    !************************************************
    ! Function    :     Initialize Variables
    ! Programmer  :     Philippe Fleischmann
    ! Date        :     2019.02.22
    !***************** ETH Zurich *******************
    !
    PROC r_RRC_InitVar()
        !
        ! Set Task on
        b_RRC_TaskReceiverOn:=TRUE;
        !
        ! Reset buffer full bits controller
        b_RRC_BufFullMa{n_RRC_R1_ChaNr}:=FALSE;
        b_RRC_BufFullMa{n_RRC_R2_ChaNr}:=FALSE;
        b_RRC_BufFullMa{n_RRC_R3_ChaNr}:=FALSE;
        b_RRC_BufFullMa{n_RRC_R4_ChaNr}:=FALSE;
        !
        ! Reset buffer full bits robot
        b_RRC_BufFullRob{n_RRC_R1_ChaNr}:=FALSE;
        b_RRC_BufFullRob{n_RRC_R2_ChaNr}:=FALSE;
        b_RRC_BufFullRob{n_RRC_R3_ChaNr}:=FALSE;
        b_RRC_BufFullRob{n_RRC_R4_ChaNr}:=FALSE;
        !
        ! Set first cycle bools
        b_RRC_FirstProtocolAfterPPMain:=TRUE;
        !
        ! Temp to measure cycle time
        b_RRC_FeedbackOut:=FALSE;
        !
        ! Reset counters controller
        n_RRC_WritePtrBufCtrl{n_RRC_R1_ChaNr}:=0;
        n_RRC_WritePtrBufCtrl{n_RRC_R2_ChaNr}:=0;
        n_RRC_WritePtrBufCtrl{n_RRC_R3_ChaNr}:=0;
        n_RRC_WritePtrBufCtrl{n_RRC_R4_ChaNr}:=0;
        !
        ! Reset counters robot
        n_RRC_WritePtrBufRob{n_RRC_R1_ChaNr}:=0;
        n_RRC_WritePtrBufRob{n_RRC_R2_ChaNr}:=0;
        n_RRC_WritePtrBufRob{n_RRC_R3_ChaNr}:=0;
        n_RRC_WritePtrBufRob{n_RRC_R4_ChaNr}:=0;
        !
        ! Clear buffer controller
        FOR i FROM 1 TO DIM(bm_RRC_RecBufferCtrl,2) DO
            !
            ! Overwrite with an empty message
            bm_RRC_RecBufferCtrl{n_RRC_R1_ChaNr,i}:=bmEmpty;
            bm_RRC_RecBufferCtrl{n_RRC_R2_ChaNr,i}:=bmEmpty;
            bm_RRC_RecBufferCtrl{n_RRC_R3_ChaNr,i}:=bmEmpty;
            bm_RRC_RecBufferCtrl{n_RRC_R4_ChaNr,i}:=bmEmpty;
            !
        ENDFOR
        !
        ! Clear buffer robots
        FOR i FROM 1 TO DIM(bm_RRC_RecBufferRob,2) DO
            !
            ! Overwrite with an empty message
            bm_RRC_RecBufferRob{n_RRC_R1_ChaNr,i}:=bmEmpty;
            bm_RRC_RecBufferRob{n_RRC_R2_ChaNr,i}:=bmEmpty;
            bm_RRC_RecBufferRob{n_RRC_R3_ChaNr,i}:=bmEmpty;
            bm_RRC_RecBufferRob{n_RRC_R4_ChaNr,i}:=bmEmpty;
            !
        ENDFOR
        !
        ! Reset expected Sequince ID
        n_RRC_SIDExpected{n_RRC_R1_ChaNr}:=0;
        n_RRC_SIDExpected{n_RRC_R2_ChaNr}:=0;
        n_RRC_SIDExpected{n_RRC_R3_ChaNr}:=0;
        n_RRC_SIDExpected{n_RRC_R4_ChaNr}:=0;
        RETURN ;
    ERROR
        ! Placeholder for Error Code...
    ENDPROC

    !************************************************
    ! Function    :     ProgError
    ! Programmer  :     Philippe Fleischmann
    ! Date        :     2019.02.22
    !***************** ETH Zurich *******************
    !
    PROC r_RRC_ProgError()
        !
        ! User Info
        TPWrite "Program Error";
        !
        ! Stop Program
        Stop;
        RETURN ;
    ERROR
        ! Placeholder for Error Code...
    ENDPROC

ENDMODULE

--- Controller Data/v2600-510970_CAADRIA/RAPID/TASK3/SYSMOD/RRC_DataTask_Rx.sys ---
MODULE RRC_DataTask_Rx(SYSMODULE)
    !***********************************************************************************
    !
    ! ETH Zurich / Robotic Fabrication Lab
    ! HIB C 13 / Stefano-Franscini-Platz 1
    ! CH-8093 Zurich
    !
    !***********************************************************************************
    !
    ! PROJECT     :  RRC - Rapid Robot Communication
    !
    ! FUNCTION    :  Includ all Task specific Data's
    !
    ! AUTHOR      :  Philippe Fleischmann
    !
    ! EMAIL       :  rrc@arch.ethz.ch
    !
    ! HISTORY     :  2019.02.22
    !
    ! Copyright   :  ETH Zurich (CH) 2019
    !                - Philippe Fleischmann
    !                - Michael Lyrenmann
    !                - Gonzalo Casas
    !
    ! License     :  This code base is governed by an EULA (End-User License Agreement)
    !                which you have received together with the software.
    !                You are not allowed to use the software on a real robots
    !                without a signed EULA.
    !
    !                A copy of the EULA content is in the controller task (T_CTRL).
    !
    !***********************************************************************************

    !************************************************
    ! Declaration :     bool
    !************************************************
    !
    CONST bool b_RRC_Run:=TRUE;
    !
    TASK PERS bool b_RRC_SocketActiv:=TRUE;
    TASK PERS bool b_RRC_PrintPrio1:=FALSE;
    TASK PERS bool b_RRC_PrintPrio2:=FALSE;
    !
    TASK PERS bool b_RRC_BufFullMa{n_RRC_NumOfCha}:=[FALSE,FALSE,FALSE,FALSE];
    TASK PERS bool b_RRC_BufFullRob{n_RRC_NumOfCha}:=[FALSE,FALSE,FALSE,FALSE];
    TASK PERS bool b_RRC_LogHelper{n_RRC_NumOfCha}:=[FALSE,FALSE,FALSE,FALSE];
    !
    TASK PERS bool b_RRC_FirstProtocolAfterPPMain:=FALSE;

    !************************************************
    ! Declaration :     num
    !************************************************
    !
    CONST num n_RRC_NumOfCha:=4;
    CONST num n_RRC_RecMinData:=49;
    CONST num n_RRC_NoOfByMsgLen:=4;
    CONST num n_RRC_TimeOutRecRobSocRec:=10;
    !
    TASK PERS num n_RRC_WritePtrBufCtrl{n_RRC_NumOfCha}:=[0,0,0,0];
    TASK PERS num n_RRC_WritePtrBufRob{n_RRC_NumOfCha}:=[1,0,0,0];
    TASK PERS num n_RRC_SIDExpected{n_RRC_NumOfCha}:=[1,0,0,0];
    TASK PERS num n_RRC_SIDIs{n_RRC_NumOfCha}:=[70001,0,0,0];
    !
    VAR num n_RRC_MsgLenRob{n_RRC_NumOfCha};
    VAR num n_RRC_NoOfRecBytesRob{n_RRC_NumOfCha};

    !************************************************
    ! Declaration :     string
    !************************************************
    !
    TASK PERS string st_RRC_EvLogMsgHeader:="RRC -- Receiver";
    TASK PERS string st_RRC_SIDRestart:="S-ID User code restarted";
    !
    TASK PERS string st_RRC_UIAnswer:="Stop";
    TASK PERS string st_RRC_ActMsg1:="Expected protocol version: 1.0";
    TASK PERS string st_RRC_ActMsg2:="Received protocol version: 2.0";
    TASK PERS string st_RRC_ActMsg3:="Expected: 2";
    TASK PERS string st_RRC_ActMsg4:="Received: 70001";
    TASK PERS string st_RRC_ActMsg5:="";
    TASK PERS string st_RRC_ActBtn1:="Stop";
    TASK PERS string st_RRC_ActBtn2:="100 mm/s";
    TASK PERS string st_RRC_ActBtn3:="Set my Speed";
    TASK PERS string st_RRC_ActBtn4:="";
    TASK PERS string st_RRC_ActBtn5:="";
    TASK PERS string st_RRC_Header:="Protocol mismatch";
    !
    VAR string st_RRC_IP_ClientRec{n_RRC_NumOfCha}:=["","","",""];

    !************************************************
    ! Declaration :     clock
    !************************************************
    !
    VAR clock clk_RRC_ReadAndUnpack;
    VAR clock clk_RRC_MsgInUntilMsgOut;

    !************************************************
    ! Declaration :     RRC_Protokol
    !************************************************
    !
    CONST RRC_Protocol pro_RRC_Empty:=[[0,0,0,0],[0,0,0,"",0,0,"",0,0,0,"",0,"",0,"",0,"",0,"",0,"",0,"",0,"",0,0,0,0,0,0,0,0,0,0,0,0,0,0,0,0,0,0,0,0,0,0,0,0,0,0,0,0,0,0,0,0,0,0,0,0,0]];
    !
    VAR RRC_Protocol pro_RRC_ActMsgRob:=[[0,0,0,0],[0,0,0,"",0,0,"",0,0,0,"",0,"",0,"",0,"",0,"",0,"",0,"",0,"",0,0,0,0,0,0,0,0,0,0,0,0,0,0,0,0,0,0,0,0,0,0,0,0,0,0,0,0,0,0,0,0,0,0,0,0,0]];
    !
    TASK PERS RRC_Protocol pro_RRC_ActMsgTemp:=[[0,0,0,0],[0,0,0,"",0,0,"",0,0,0,"",0,"",0,"",0,"",0,"",0,"",0,"",0,"",0,0,0,0,0,0,0,0,0,0,0,0,0,0,0,0,0,0,0,0,0,0,0,0,0,0,0,0,0,0,0,0,0,0,0,0,0]];
    !
    TASK PERS RRC_Protocol pro_RRC_ActMsgRec{n_RRC_NumOfCha}:=[
    [[91,2,1.77453E+9,955],[1,0,15,"r_RRC_PrintText",1,0,"",0,1,24,"Welcome to COMPAS_RRC On",0,"",0,"",0,"",0,"",0,"",0,"",0,"",0,0,0,0,0,0,0,0,0,0,0,0,0,0,0,0,0,0,0,0,0,0,0,0,0,0,0,0,0,0,0,0,0,0,0,0,0]],
    [[67,4,1.58281E+9,242],[4,0,15,"r_RRC_WaitTime",1,0,"",0,0,24,"E-Level Channel 2 Controller",0,"",0,"",0,"",0,"",0,"",0,"",0,"",1,1,0,0,0,0,0,0,0,0,0,0,0,0,0,0,0,0,0,0,0,0,0,0,0,0,0,0,0,0,0,0,0,0,0,0,0]],
    [[120,4,1.55775E+9,695],[11,0,12,"r_RRC_MoveL",1,0,"",0,0,0,"",0,"",0,"",0,"",0,"",0,"",0,"",0,"",15,542.04,-200,237.57,0,0,1,0,28000,-3400,-3138,0,0,0,230,20,0,0,0,0,0,0,0,0,0,0,0,0,0,0,0,0,0,0,0,0,0]],
    [[120,4,1.55775E+9,695],[11,0,12,"r_RRC_MoveL",1,0,"",0,0,0,"",0,"",0,"",0,"",0,"",0,"",0,"",0,"",15,542.04,-200,237.57,0,0,1,0,28000,-3400,-3138,0,0,0,230,20,0,0,0,0,0,0,0,0,0,0,0,0,0,0,0,0,0,0,0,0,0]]];

    !************************************************
    ! Declaration :     rawbytes
    !************************************************
    !
    VAR rawbytes rb_RRC_BufferMsgLenRob{n_RRC_NumOfCha};
    VAR rawbytes rb_RRC_BufferRob{n_RRC_NumOfCha};

    !************************************************
    ! Declaration :     socketdev
    !************************************************
    !
    VAR socketdev sod_RRC_ServerRec{n_RRC_NumOfCha};
    VAR socketdev sod_RRC_ClientRec{n_RRC_NumOfCha};

    !************************************************
    ! Declaration :     RRC_buffer_msg
    !************************************************
    !
    CONST RRC_buffer_msg bmEmpty:=[[0,0,0,"",0,0,"",0,0,0,"",0,"",0,"",0,"",0,"",0,"",0,"",0,"",0,0,0,0,0,0,0,0,0,0,0,0,0,0,0,0,0,0,0,0,0,0,0,0,0,0,0,0,0,0,0,0,0,0,0,0,0],FALSE];
ENDMODULE

--- Controller Data/v2600-510970_CAADRIA/RAPID/TASK3/SYSMOD/RRC_Log_Rx.sys ---
MODULE RRC_Log_Rx(SYSMODULE)
    !***********************************************************************************
    !
    ! ETH Zurich / Robotic Fabrication Lab
    ! HIB C 13 / Stefano-Franscini-Platz 1
    ! CH-8093 Zurich
    !
    !***********************************************************************************
    !
    ! PROJECT     :  RRC - Rapid Robot Communication
    !
    ! FUNCTION    :  Inclouds all logger functions
    !
    ! AUTHOR      :  Philippe Fleischmann
    !
    ! EMAIL       :  rrc@arch.ethz.ch
    !
    ! HISTORY     :  2019.02.22
    !
    ! Copyright   :  ETH Zurich (CH) 2019
    !                - Philippe Fleischmann
    !                - Michael Lyrenmann
    !                - Gonzalo Casas
    !
    ! License     :  This code base is governed by an EULA (End-User License Agreement)
    !                which you have received together with the software.
    !                You are not allowed to use the software on a real robots
    !                without a signed EULA.
    !
    !                A copy of the EULA content is in the controller task (T_CTRL).
    !
    !***********************************************************************************

    !************************************************
    ! Declaration :     bool
    !************************************************
    !
    CONST bool b_RRC_LogActiv:=TRUE;

    !************************************************
    ! Declaration :     num
    !************************************************
    !
    TASK PERS num n_RRC_LogMsgCountr:=0;
    TASK PERS num n_RRC_FileNr:=1;
    CONST num n_RRC_LogMaxMsg:=1000000;

    !************************************************
    ! Declaration :     string
    !************************************************
    !
    CONST string st_RRC_LogDirPathRC:="RemovableDisk1:RRC_Log/";
    CONST string st_RRC_LogDirPathVC:="Home:/RRC_Log/";
    TASK PERS string st_RRC_LogDirPath:="RemovableDisk1:RRC_Log/";
    CONST string st_RRC_LogFileName:="RRC_LogReceiver";
    CONST string st_RRC_LogFileFormat:=".csv";
    CONST string st_RRC_LogProgrammer:="Philipppe Fleischmann";
    !
    CONST string stTab:="\09";

    ! Global System Data
    TASK PERS string st_RFL_SystemDate:="2018-06-28";
    TASK PERS string st_RFL_SystemTime:="15:49:26";

    !************************************************
    ! Declaration :     iodev
    !************************************************
    !
    VAR iodev iodev_RRC_LogFile;

    !************************************************
    ! Declaration :     dir
    !************************************************
    !
    VAR dir dir_RRC_Dev;

    !************************************************
    ! Declaration :     clock
    !************************************************
    !
    VAR clock ck_RRC_LogTimer;

    !************************************************
    ! Discription :     Steps for log integration in code
    ! Programmer  :     Philippe Fleischmann
    ! Date        :     2019.02.22
    !***************** ETH Zurich *******************
    !
    ! 1. Create a log folder, run the procedure manuali PP to Routine
    !* r_RRC_CrateLogFolder;
    !
    ! 2. Integrate Initialzie log function
    !* r_RRC_LogInit
    !
    ! 3. Integrate write log
    !* IF b_RRC_LogActiv=TRUE r_RRC_LogWriteRhinoMsg message_command;
    !
    ! 4. Integrate Close file (when posible)
    !* IF b_RRC_LogActiv=TRUE r_RRC_LogFileClose;
    !
    !************************************************

    !************************************************
    ! Function    :     Log initialization
    ! Programmer  :     Philippe Fleischmann
    ! Date        :     2019.02.22
    !***************** ETH Zurich *******************
    !
    PROC r_RRC_LogTest()
        !
        ! Initialize logfile
        r_RRC_LogProtInit;
        !
        ! Load protocol message
        ! Header
        pro_RRC_ActMsgRob.ProtocolHeader.M_Len:=104;
        pro_RRC_ActMsgRob.ProtocolHeader.Ver:=1;
        pro_RRC_ActMsgRob.ProtocolHeader.TS_Sec:=33;
        pro_RRC_ActMsgRob.ProtocolHeader.TS_NSec:=399;
        !
        ! Main data
        pro_RRC_ActMsgRob.ProtocolData.S_ID:=300;
        pro_RRC_ActMsgRob.ProtocolData.E_Lev:=0;
        pro_RRC_ActMsgRob.ProtocolData.F_Lev:=1;
        pro_RRC_ActMsgRob.ProtocolData.I_Len:=8;
        pro_RRC_ActMsgRob.ProtocolData.Instr:="MoveAbsJ";
        pro_RRC_ActMsgRob.ProtocolData.F_Len:=4;
        pro_RRC_ActMsgRob.ProtocolData.Feedb:="Done";
        pro_RRC_ActMsgRob.ProtocolData.F_ID:=300;
        !
        ! String parameter
        pro_RRC_ActMsgRob.ProtocolData.St_Cnt:=5;
        pro_RRC_ActMsgRob.ProtocolData.St1_Len:=4;
        pro_RRC_ActMsgRob.ProtocolData.St1:="This";
        pro_RRC_ActMsgRob.ProtocolData.St2_Len:=2;
        pro_RRC_ActMsgRob.ProtocolData.St2:="is";
        pro_RRC_ActMsgRob.ProtocolData.St3_Len:=1;
        pro_RRC_ActMsgRob.ProtocolData.St3:="a";
        pro_RRC_ActMsgRob.ProtocolData.St4_Len:=8;
        pro_RRC_ActMsgRob.ProtocolData.St4:="protocol";
        pro_RRC_ActMsgRob.ProtocolData.St5_Len:=5;
        pro_RRC_ActMsgRob.ProtocolData.St5:="test";
        !
        ! Value parameter
        pro_RRC_ActMsgRob.ProtocolData.V_Cnt:=1;
        pro_RRC_ActMsgRob.ProtocolData.V1:=99;
        FOR i FROM 1 TO 1 DO


            r_RRC_LogPro pro_RRC_ActMsgRob;

        ENDFOR

        Close iodev_RRC_LogFile;

        Stop;

        RETURN ;
    ERROR
    ENDPROC

    !************************************************
    ! Function    :     Initialize protocol log
    ! Programmer  :     Philippe Fleischmann
    ! Date        :     2019.02.22
    !***************** ETH Zurich *******************
    !
    PROC r_RRC_LogProtInit()
        !
        ! Selcet the writ path for the log file
        IF RobOS()=TRUE THEN
            !
            ! Real controller write to MemoryStick
            st_RRC_LogDirPath:=st_RRC_LogDirPathRC;
        ELSE
            !
            ! Virtual controller write to Home
            st_RRC_LogDirPath:=st_RRC_LogDirPathVC;
        ENDIF
        !
        ! Initalize variables
        n_RRC_LogMsgCountr:=0;
        !
        ! Opent directory
        OpenDir dir_RRC_Dev,st_RRC_LogDirPath;
        !
        ! Check for log file
        IF IsFile(st_RRC_LogDirPath+st_RRC_LogFileName+st_RRC_LogFileFormat) THEN
            !
            ! Remove the old log file
            RemoveFile st_RRC_LogDirPath+st_RRC_LogFileName+st_RRC_LogFileFormat;
        ENDIF
        !
        ! Create and open a new log file
        Open st_RRC_LogDirPath+st_RRC_LogFileName+st_RRC_LogFileFormat,iodev_RRC_LogFile\Write;
        !
        ! Write column title for
        Write iodev_RRC_LogFile,"L-Nr;LogTime;LogFormat;"\NoNewLine;
        Write iodev_RRC_LogFile,"M_Len;Ver;TS-Sec;TS-NSec;"\NoNewLine;
        Write iodev_RRC_LogFile,"S_ID;E_Lev;I_Len;Instr;F_Lev;F_Len;Feedb;F_ID;"\NoNewLine;
        Write iodev_RRC_LogFile,"St_Ctr;St1_Len;St1;St2_Len;St2;St3_Len;St3;St4_Len;St4;St5_Len;St5;"\NoNewLine;
        Write iodev_RRC_LogFile,"V_Ctr;V1;V2;V3;V4;V5;V6;V7;V8;V9;V10;"\NoNewLine;
        Write iodev_RRC_LogFile,"V11;V12;V13;V14;V15;V16;V17;V18;V19;V20;"\NoNewLine;
        Write iodev_RRC_LogFile,"V21;V22;V23;V24;V25;V26;V27;V28;V29;V30;";
        !
        ! Reset and start log timer
        ClkReset ck_RRC_LogTimer;
        ClkStart ck_RRC_LogTimer;
        !
        ! Log message
        r_RRC_EvLogMsg st_RRC_LogFileName,"Log inititalizaion, done";
        RETURN ;
    ERROR
        !
        ! Handle error open directory
        IF ERRNO=ERR_FILEACC THEN
            !
            ! Create the log folder
            MakeDir st_RRC_LogDirPath;
            !
            ! Log message
            r_RRC_EvLogMsg st_RRC_LogFileName,"Log Directory created";
            !
            ! Retyry to open directory
            RETRY;
        ENDIF
        Stop;
        Stop;
    ENDPROC

    !************************************************
    ! Function    :     Log protocol
    ! Programmer  :     Philippe Fleischmann
    ! Date        :     2019.02.22
    !***************** ETH Zurich *******************
    !
    PROC r_RRC_LogPro(RRC_Protocol proMsg)
        !
        ! Increuse log message counter
        Incr n_RRC_LogMsgCountr;
        !
        ! Log only until max message is reached
        IF n_RRC_LogMsgCountr<=n_RRC_LogMaxMsg THEN
            !
            ! Add counter nuber and time
            Write iodev_RRC_LogFile,NumToStr(n_RRC_LogMsgCountr,0)+";"\NoNewLine;
            Write iodev_RRC_LogFile,NumToStr(ClkRead(ck_RRC_LogTimer\HighRes),3)+";"\NoNewLine;
            !
            ! Add log format
            Write iodev_RRC_LogFile,"protocol"+";"\NoNewLine;
            !
            ! Add protocol header
            Write iodev_RRC_LogFile,NumToStr(proMsg.ProtocolHeader.M_Len,0)+";"\NoNewLine;
            Write iodev_RRC_LogFile,NumToStr(proMsg.ProtocolHeader.Ver,0)+";"\NoNewLine;
            Write iodev_RRC_LogFile,NumToStr(proMsg.ProtocolHeader.TS_Sec,0)+";"\NoNewLine;
            Write iodev_RRC_LogFile,NumToStr(proMsg.ProtocolHeader.TS_NSec,3)+";"\NoNewLine;
            !
            ! Protocol main data
            Write iodev_RRC_LogFile,NumToStr(proMsg.ProtocolData.S_ID,0)+";"\NoNewLine;
            Write iodev_RRC_LogFile,NumToStr(proMsg.ProtocolData.E_Lev,0)+";"\NoNewLine;
            Write iodev_RRC_LogFile,NumToStr(proMsg.ProtocolData.I_Len,0)+";"\NoNewLine;
            Write iodev_RRC_LogFile,proMsg.ProtocolData.Instr+";"\NoNewLine;
            Write iodev_RRC_LogFile,NumToStr(proMsg.ProtocolData.F_Lev,0)+";"\NoNewLine;
            Write iodev_RRC_LogFile,NumToStr(proMsg.ProtocolData.F_Len,0)+";"\NoNewLine;
            Write iodev_RRC_LogFile,proMsg.ProtocolData.Feedb+";"\NoNewLine;
            Write iodev_RRC_LogFile,NumToStr(proMsg.ProtocolData.F_ID,0)+";"\NoNewLine;
            !
            ! Protocol string parameter
            Write iodev_RRC_LogFile,NumToStr(proMsg.ProtocolData.St_Cnt,0)+";"\NoNewLine;
            Write iodev_RRC_LogFile,NumToStr(proMsg.ProtocolData.St1_Len,0)+";"\NoNewLine;
            Write iodev_RRC_LogFile,proMsg.ProtocolData.St1+";"\NoNewLine;
            Write iodev_RRC_LogFile,NumToStr(proMsg.ProtocolData.St2_Len,0)+";"\NoNewLine;
            Write iodev_RRC_LogFile,proMsg.ProtocolData.St2+";"\NoNewLine;
            Write iodev_RRC_LogFile,NumToStr(proMsg.ProtocolData.St3_Len,0)+";"\NoNewLine;
            Write iodev_RRC_LogFile,proMsg.ProtocolData.St3+";"\NoNewLine;
            Write iodev_RRC_LogFile,NumToStr(proMsg.ProtocolData.St4_Len,0)+";"\NoNewLine;
            Write iodev_RRC_LogFile,proMsg.ProtocolData.St4+";"\NoNewLine;
            Write iodev_RRC_LogFile,NumToStr(proMsg.ProtocolData.St5_Len,0)+";"\NoNewLine;
            Write iodev_RRC_LogFile,proMsg.ProtocolData.St5+";"\NoNewLine;
            !
            ! Protocol value parameter
            Write iodev_RRC_LogFile,NumToStr(proMsg.ProtocolData.V_Cnt,0)+";"\NoNewLine;
            Write iodev_RRC_LogFile,NumToStr(proMsg.ProtocolData.V1,3)+";"\NoNewLine;
            Write iodev_RRC_LogFile,NumToStr(proMsg.ProtocolData.V2,3)+";"\NoNewLine;
            Write iodev_RRC_LogFile,NumToStr(proMsg.ProtocolData.V3,3)+";"\NoNewLine;
            Write iodev_RRC_LogFile,NumToStr(proMsg.ProtocolData.V4,3)+";"\NoNewLine;
            Write iodev_RRC_LogFile,NumToStr(proMsg.ProtocolData.V5,3)+";"\NoNewLine;
            Write iodev_RRC_LogFile,NumToStr(proMsg.ProtocolData.V6,3)+";"\NoNewLine;
            Write iodev_RRC_LogFile,NumToStr(proMsg.ProtocolData.V7,3)+";"\NoNewLine;
            Write iodev_RRC_LogFile,NumToStr(proMsg.ProtocolData.V8,3)+";"\NoNewLine;
            Write iodev_RRC_LogFile,NumToStr(proMsg.ProtocolData.V9,3)+";"\NoNewLine;
            Write iodev_RRC_LogFile,NumToStr(proMsg.ProtocolData.V10,3)+";"\NoNewLine;
            Write iodev_RRC_LogFile,NumToStr(proMsg.ProtocolData.V11,3)+";"\NoNewLine;
            Write iodev_RRC_LogFile,NumToStr(proMsg.ProtocolData.V12,3)+";"\NoNewLine;
            Write iodev_RRC_LogFile,NumToStr(proMsg.ProtocolData.V13,3)+";"\NoNewLine;
            Write iodev_RRC_LogFile,NumToStr(proMsg.ProtocolData.V14,3)+";"\NoNewLine;
            Write iodev_RRC_LogFile,NumToStr(proMsg.ProtocolData.V15,3)+";"\NoNewLine;
            Write iodev_RRC_LogFile,NumToStr(proMsg.ProtocolData.V16,3)+";"\NoNewLine;
            Write iodev_RRC_LogFile,NumToStr(proMsg.ProtocolData.V17,3)+";"\NoNewLine;
            Write iodev_RRC_LogFile,NumToStr(proMsg.ProtocolData.V18,3)+";"\NoNewLine;
            Write iodev_RRC_LogFile,NumToStr(proMsg.ProtocolData.V19,3)+";"\NoNewLine;
            Write iodev_RRC_LogFile,NumToStr(proMsg.ProtocolData.V20,3)+";"\NoNewLine;
            Write iodev_RRC_LogFile,NumToStr(proMsg.ProtocolData.V21,3)+";"\NoNewLine;
            Write iodev_RRC_LogFile,NumToStr(proMsg.ProtocolData.V22,3)+";"\NoNewLine;
            Write iodev_RRC_LogFile,NumToStr(proMsg.ProtocolData.V23,3)+";"\NoNewLine;
            Write iodev_RRC_LogFile,NumToStr(proMsg.ProtocolData.V24,3)+";"\NoNewLine;
            Write iodev_RRC_LogFile,NumToStr(proMsg.ProtocolData.V25,3)+";"\NoNewLine;
            Write iodev_RRC_LogFile,NumToStr(proMsg.ProtocolData.V26,3)+";"\NoNewLine;
            Write iodev_RRC_LogFile,NumToStr(proMsg.ProtocolData.V27,3)+";"\NoNewLine;
            Write iodev_RRC_LogFile,NumToStr(proMsg.ProtocolData.V28,3)+";"\NoNewLine;
            Write iodev_RRC_LogFile,NumToStr(proMsg.ProtocolData.V29,3)+";"\NoNewLine;
            Write iodev_RRC_LogFile,NumToStr(proMsg.ProtocolData.V30,3)+";"\NoNewLine;
            !
            ! Protocol end
            Write iodev_RRC_LogFile,";";
        ENDIF


        RETURN ;
    ERROR
        ! Placeholder for Error Code...
    ENDPROC

ENDMODULE

--- Controller Data/v2600-510970_CAADRIA/RAPID/TASK4/SYSMOD/RRC_Control_Tx.sys ---
MODULE RRC_Control_Tx(SYSMODULE)
    !***********************************************************************************
    !
    ! ETH Zurich / Robotic Fabrication Lab
    ! HIB C 13 / Stefano-Franscini-Platz 1
    ! CH-8093 Zurich
    !
    !***********************************************************************************
    !
    ! PROJECT     :  RRC - Rapid Robot Communication
    !
    ! FUNCTION    :  Control modul for the project
    !
    ! AUTHOR      :  Philippe Fleischmann
    !
    ! EMAIL       :  rrc@arch.ethz.ch
    !
    ! HISTORY     :  2019.02.22
    !
    ! Copyright   :  ETH Zurich (CH) 2019
    !                - Philippe Fleischmann
    !                - Michael Lyrenmann
    !                - Gonzalo Casas
    !
    ! License     :  This code base is governed by an EULA (End-User License Agreement)
    !                which you have received together with the software.
    !                You are not allowed to use the software on a real robots
    !                without a signed EULA.
    !
    !                A copy of the EULA content is in the controller task (T_CTRL).
    !
    !***********************************************************************************

    !************************************************
    ! Function    :     Main for Project RRC
    ! Programmer  :     Philippe Fleischmann
    ! Date        :     2019.02.22
    !***************** ETH Zurich *******************
    !
    PROC r_RRC_Main()
        !
        ! Wait until controller has set taskliste all
        WaitTime n_RRC_TimeTaskLiAll;
        !
        ! Task synchronisation
        WaitSyncTask id_RRC_MainSta,tl_RRC_All;
        !
        ! Message for Operator
        TPWrite "RRC Main";
        !
        ! Inititalize cell
        r_RRC_InitCell;
        !
        ! Work process
        WHILE b_RRC_Run=TRUE DO
            !
            ! Check and send data to client
            IF b_RRC_Com{n_RRC_R1_ChaNr}=TRUE THEN
                !
                ! For robot
                IF bm_RRC_SenBufferRob{n_RRC_R1_ChaNr,n_RRC_ReadPtrSenBufRob{n_RRC_R1_ChaNr}}.startbit=TRUE r_RRC_PackSendDataToClient\Rob,n_RRC_R1_ChaNr;
                !
                ! For controller
                IF bm_RRC_SenBufferCtrl{n_RRC_R1_ChaNr,n_RRC_ReadPtrSenBufCtrl{n_RRC_R1_ChaNr}}.startbit=TRUE r_RRC_PackSendDataToClient\Ctrl,n_RRC_R1_ChaNr;
            ENDIF
            !
            ! Check and send data to client
            IF b_RRC_Com{n_RRC_R2_ChaNr}=TRUE THEN
                !
                ! For robot
                IF bm_RRC_SenBufferRob{n_RRC_R2_ChaNr,n_RRC_ReadPtrSenBufRob{n_RRC_R2_ChaNr}}.startbit=TRUE r_RRC_PackSendDataToClient\Rob,n_RRC_R2_ChaNr;
                !
                ! For controller
                IF bm_RRC_SenBufferCtrl{n_RRC_R2_ChaNr,n_RRC_ReadPtrSenBufCtrl{n_RRC_R2_ChaNr}}.startbit=TRUE r_RRC_PackSendDataToClient\Ctrl,n_RRC_R2_ChaNr;
            ENDIF
            !
            ! Check and send data to client
            IF b_RRC_Com{n_RRC_R3_ChaNr}=TRUE THEN
                !
                ! For robot
                IF bm_RRC_SenBufferRob{n_RRC_R3_ChaNr,n_RRC_ReadPtrSenBufRob{n_RRC_R3_ChaNr}}.startbit=TRUE r_RRC_PackSendDataToClient\Rob,n_RRC_R3_ChaNr;
                !
                ! For controller
                IF bm_RRC_SenBufferCtrl{n_RRC_R3_ChaNr,n_RRC_ReadPtrSenBufCtrl{n_RRC_R3_ChaNr}}.startbit=TRUE r_RRC_PackSendDataToClient\Ctrl,n_RRC_R3_ChaNr;
            ENDIF
            !
            ! Check and send data to client
            IF b_RRC_Com{n_RRC_R4_ChaNr}=TRUE THEN
                !
                ! For robot
                IF bm_RRC_SenBufferRob{n_RRC_R4_ChaNr,n_RRC_ReadPtrSenBufRob{n_RRC_R4_ChaNr}}.startbit=TRUE r_RRC_PackSendDataToClient\Rob,n_RRC_R4_ChaNr;
                !
                ! For controller
                IF bm_RRC_SenBufferCtrl{n_RRC_R4_ChaNr,n_RRC_ReadPtrSenBufCtrl{n_RRC_R4_ChaNr}}.startbit=TRUE r_RRC_PackSendDataToClient\Ctrl,n_RRC_R4_ChaNr;
            ENDIF
        ENDWHILE
        !
        ! Message for Operator
        TPWrite "RRC End";
        !
        ! Task synchronisation
        WaitSyncTask id_RRC_MainEnd,tl_RRC_All;
        !
        RETURN ;
    ERROR
        ! Placeholder for Error Code...
    ENDPROC

    !************************************************
    ! Function    :     Initialize Cell
    ! Programmer  :     Philippe Fleischmann
    ! Date        :     2019.02.22
    !***************** ETH Zurich *******************
    !
    PROC r_RRC_InitCell()
        !
        ! Task synchronisation
        WaitSyncTask id_RRC_InitSta,tl_RRC_All;
        !
        ! Task synchronisation wait for controller data
        WaitSyncTask id_RRC_InitCtrl,tl_RRC_All;
        !
        ! Initialize variables
        r_RRC_InitVar;
        !
        ! Initialize sockets
        IF b_RRC_SocketActiv=TRUE r_RRC_InitSockets;
        !
        ! Task synchronisation
        WaitSyncTask id_RRC_InitEnd,tl_RRC_All;
        RETURN ;
    ERROR
        ! Placeholder for Error Code...
    ENDPROC

    !************************************************
    ! Function    :     Initialize Variables
    ! Programmer  :     Philippe Fleischmann
    ! Date        :     2019.02.22
    !***************** ETH Zurich *******************
    !
    PROC r_RRC_InitVar()
        !
        ! Set Task on
        b_RRC_TaskSenderOn:=TRUE;
        !
        ! Reset and start timestamp
        ClkReset clk_RRC_TimeStamp;
        ClkStart clk_RRC_TimeStamp;
        !
        ! Reset Counters
        n_RRC_WritePtrSenBufCtrl{n_RRC_R1_ChaNr}:=0;
        n_RRC_WritePtrSenBufCtrl{n_RRC_R2_ChaNr}:=0;
        n_RRC_WritePtrSenBufCtrl{n_RRC_R3_ChaNr}:=0;
        n_RRC_WritePtrSenBufCtrl{n_RRC_R4_ChaNr}:=0;
        !
        n_RRC_WritePtrSenBufRob{n_RRC_R1_ChaNr}:=0;
        n_RRC_WritePtrSenBufRob{n_RRC_R2_ChaNr}:=0;
        n_RRC_WritePtrSenBufRob{n_RRC_R3_ChaNr}:=0;
        n_RRC_WritePtrSenBufRob{n_RRC_R4_ChaNr}:=0;
        !
        n_RRC_ReadPtrSenBufCtrl{n_RRC_R1_ChaNr}:=1;
        n_RRC_ReadPtrSenBufCtrl{n_RRC_R2_ChaNr}:=1;
        n_RRC_ReadPtrSenBufCtrl{n_RRC_R3_ChaNr}:=1;
        n_RRC_ReadPtrSenBufCtrl{n_RRC_R4_ChaNr}:=1;
        !
        n_RRC_ReadPtrSenBufRob{n_RRC_R1_ChaNr}:=1;
        n_RRC_ReadPtrSenBufRob{n_RRC_R2_ChaNr}:=1;
        n_RRC_ReadPtrSenBufRob{n_RRC_R3_ChaNr}:=1;
        n_RRC_ReadPtrSenBufRob{n_RRC_R4_ChaNr}:=1;
        !
        n_RRC_SenHeaderSqzNr{n_RRC_R1_ChaNr}:=0;
        n_RRC_SenHeaderSqzNr{n_RRC_R2_ChaNr}:=0;
        n_RRC_SenHeaderSqzNr{n_RRC_R3_ChaNr}:=0;
        n_RRC_SenHeaderSqzNr{n_RRC_R4_ChaNr}:=0;
        !
        ! Clear Buffers
        FOR i FROM 1 TO DIM(bm_RRC_SenBufferCtrl,2) DO
            !
            ! Overwrite with an empty message
            bm_RRC_SenBufferCtrl{n_RRC_R1_ChaNr,i}:=bmEmpty;
            bm_RRC_SenBufferCtrl{n_RRC_R2_ChaNr,i}:=bmEmpty;
            bm_RRC_SenBufferCtrl{n_RRC_R3_ChaNr,i}:=bmEmpty;
            bm_RRC_SenBufferCtrl{n_RRC_R4_ChaNr,i}:=bmEmpty;
        ENDFOR
        !
        ! Clear Buffers
        FOR i FROM 1 TO DIM(bm_RRC_SenBufferRob,2) DO
            !
            ! Overwrite with an empty message
            bm_RRC_SenBufferRob{n_RRC_R1_ChaNr,i}:=bmEmpty;
            bm_RRC_SenBufferRob{n_RRC_R2_ChaNr,i}:=bmEmpty;
            bm_RRC_SenBufferRob{n_RRC_R3_ChaNr,i}:=bmEmpty;
            bm_RRC_SenBufferRob{n_RRC_R4_ChaNr,i}:=bmEmpty;
        ENDFOR
        !
        ! Clear Buffers
        FOR i FROM 1 TO DIM(pro_RRC_ActMsgSen,2) DO
            !
            ! Overwrite with an empty protocol
            pro_RRC_ActMsgSen{1,i}:=proEmpty;
            pro_RRC_ActMsgSen{1,i}:=proEmpty;
            pro_RRC_ActMsgSen{1,i}:=proEmpty;
            pro_RRC_ActMsgSen{1,i}:=proEmpty;
            !
            pro_RRC_ActMsgSen{2,i}:=proEmpty;
            pro_RRC_ActMsgSen{2,i}:=proEmpty;
            pro_RRC_ActMsgSen{2,i}:=proEmpty;
            pro_RRC_ActMsgSen{2,i}:=proEmpty;
        ENDFOR
        RETURN ;
    ERROR
        ! Placeholder for Error Code...
    ENDPROC

    !************************************************
    ! Function    :     ProgError
    ! Programmer  :     Philippe Fleischmann
    ! Date        :     2019.02.22
    !***************** ETH Zurich *******************
    !
    PROC r_RRC_ProgError()
        !
        ! User Info
        TPWrite "Program Error";
        !
        ! Stop Program
        Stop;
        RETURN ;
    ERROR
        ! Placeholder for Error Code...
    ENDPROC

ENDMODULE

--- Controller Data/v2600-510970_CAADRIA/RAPID/TASK4/SYSMOD/RRC_DataTask_Tx.sys ---
MODULE RRC_DataTask_Tx(SYSMODULE)
    !***********************************************************************************
    !
    ! ETH Zurich / Robotic Fabrication Lab
    ! HIB C 13 / Stefano-Franscini-Platz 1
    ! CH-8093 Zurich
    !
    !***********************************************************************************
    !
    ! PROJECT     :  RRC - Rapid Robot Communication
    !
    ! FUNCTION    :  Includ all Task specific Data's
    !
    ! AUTHOR      :  Philippe Fleischmann
    !
    ! EMAIL       :  rrc@arch.ethz.ch
    !
    ! HISTORY     :  2019.02.22
    !
    ! Copyright   :  ETH Zurich (CH) 2019
    !                - Philippe Fleischmann
    !                - Michael Lyrenmann
    !                - Gonzalo Casas
    !
    ! License     :  This code base is governed by an EULA (End-User License Agreement)
    !                which you have received together with the software.
    !                You are not allowed to use the software on a real robots
    !                without a signed EULA.
    !
    !                A copy of the EULA content is in the controller task (T_CTRL).
    !
    !***********************************************************************************

    !************************************************
    ! Declaration :     bool
    !************************************************
    !
    CONST bool b_RRC_Run:=TRUE;
    !
    TASK PERS bool b_RRC_PrintPrio1:=FALSE;
    !
    TASK PERS bool b_RRC_SocketActiv:=TRUE;

    !************************************************
    ! Declaration :     num
    !************************************************
    !
    CONST num n_RRC_NumOfCha:=4;
    CONST num n_RRC_SenMinData:=1;
    CONST num n_RRC_NoOfByMsgLen:=4;
    CONST num n_RRC_SenHeaderMaxSqzNrRob:=1000000;
    CONST num n_RRC_ProtocolCtrl:=1;
    CONST num n_RRC_ProtocolRob:=2;
    CONST num n_RRC_SendProtocolPerChannel:=2;
    !
    TASK PERS num n_RRC_ReadPtrSenBufRob{n_RRC_NumOfCha}:=[2,1,1,1];
    TASK PERS num n_RRC_ReadPtrSenBufCtrl{n_RRC_NumOfCha}:=[1,1,1,1];
    !
    TASK PERS num n_RRC_SenHeaderSqzNr{n_RRC_NumOfCha}:=[1,0,0,0];
    !
    TASK PERS num n_RRC_SenMsgLenRob:=63;
    !
    TASK PERS num n_RRC_TimeStamp:=77.719;
    TASK PERS num n_RRC_TimeStampSec:=77;
    TASK PERS num n_RRC_TimeStampNanoSec:=719;

    !************************************************
    ! Declaration :     string
    !************************************************
    !
    TASK PERS string st_RRC_EvLogMsgHeader:="RRC -- Sender";
    !
    VAR string st_RRC_IP_ClientSen{n_RRC_NumOfCha}:=["","","",""];

    !************************************************
    ! Declaration :     clock
    !************************************************
    !
    VAR clock clk_RRC_TimeStamp;
    VAR clock clk_RRC_PackAndSend;

    !************************************************
    ! Declaration :     socketdev
    !************************************************
    !
    TASK VAR socketdev sod_RRC_ServerSen{n_RRC_NumOfCha};
    TASK VAR socketdev sod_RRC_ClientSen{n_RRC_NumOfCha};

    !************************************************
    ! Declaration :     RRC_Protokol
    !************************************************
    !
    CONST RRC_Protocol proEmpty:=[[0,0,0,0],[0,0,0,"",0,0,"",0,0,0,"",0,"",0,"",0,"",0,"",0,"",0,"",0,"",0,0,0,0,0,0,0,0,0,0,0,0,0,0,0,0,0,0,0,0,0,0,0,0,0,0,0,0,0,0,0,0,0,0,0,0,0]];
    !
    !* TASK VAR RRC_Protocol pro_RRC_ActMsgRob:=[[0,0,0,0],[0,0,0,"",0,0,"",0,0,0,"",0,"",0,"",0,"",0,"",0,0,0,0,0,0,0,0,0,0,0,0,0,0,0,0,0,0,0,0,0,0,0,0,0,0,0,0,0,0,0]];
    !
    TASK PERS RRC_Protocol pro_RRC_ActMsgSen{n_RRC_SendProtocolPerChannel,n_RRC_NumOfCha}:=[
    [[[0,0,0,0],[0,0,0,"",0,0,"",0,0,0,"",0,"",0,"",0,"",0,"",0,"",0,"",0,"",0,0,0,0,0,0,0,0,0,0,0,0,0,0,0,0,0,0,0,0,0,0,0,0,0,0,0,0,0,0,0,0,0,0,0,0,0]],
    [[0,0,0,0],[0,0,0,"",0,0,"",0,0,0,"",0,"",0,"",0,"",0,"",0,"",0,"",0,"",0,0,0,0,0,0,0,0,0,0,0,0,0,0,0,0,0,0,0,0,0,0,0,0,0,0,0,0,0,0,0,0,0,0,0,0,0]],
    [[0,0,0,0],[0,0,0,"",0,0,"",0,0,0,"",0,"",0,"",0,"",0,"",0,"",0,"",0,"",0,0,0,0,0,0,0,0,0,0,0,0,0,0,0,0,0,0,0,0,0,0,0,0,0,0,0,0,0,0,0,0,0,0,0,0,0]],
    [[0,0,0,0],[0,0,0,"",0,0,"",0,0,0,"",0,"",0,"",0,"",0,"",0,"",0,"",0,"",0,0,0,0,0,0,0,0,0,0,0,0,0,0,0,0,0,0,0,0,0,0,0,0,0,0,0,0,0,0,0,0,0,0,0,0,0]]],

    [[[67,2,77,719],[1,0,15,"r_RRC_PrintText",0,4,"Done",1,0,0,"",0,"",0,"",0,"",0,"",0,"",0,"",0,"",0,0,0,0,0,0,0,0,0,0,0,0,0,0,0,0,0,0,0,0,0,0,0,0,0,0,0,0,0,0,0,0,0,0,0,0,0]],
    [[0,0,0,0],[0,0,0,"",0,0,"",0,0,0,"",0,"",0,"",0,"",0,"",0,"",0,"",0,"",0,0,0,0,0,0,0,0,0,0,0,0,0,0,0,0,0,0,0,0,0,0,0,0,0,0,0,0,0,0,0,0,0,0,0,0,0]],
    [[0,0,0,0],[0,0,0,"",0,0,"",0,0,0,"",0,"",0,"",0,"",0,"",0,"",0,"",0,"",0,0,0,0,0,0,0,0,0,0,0,0,0,0,0,0,0,0,0,0,0,0,0,0,0,0,0,0,0,0,0,0,0,0,0,0,0]],
    [[0,0,0,0],[0,0,0,"",0,0,"",0,0,0,"",0,"",0,"",0,"",0,"",0,"",0,"",0,"",0,0,0,0,0,0,0,0,0,0,0,0,0,0,0,0,0,0,0,0,0,0,0,0,0,0,0,0,0,0,0,0,0,0,0,0,0]]]];

    !************************************************
    ! Declaration :     rawbytes
    !************************************************
    !
    TASK VAR rawbytes rb_RRC_SenTempBuffer;
    TASK VAR rawbytes rb_RRC_SenBufferMsgLen;
    TASK VAR rawbytes rb_RRC_SenBuffer;

    !************************************************
    ! Declaration :     RRC_buffer_msg
    !************************************************
    !
    CONST RRC_buffer_msg bmEmpty:=[[0,0,0,"",0,0,"",0,0,0,"",0,"",0,"",0,"",0,"",0,"",0,"",0,"",0,0,0,0,0,0,0,0,0,0,0,0,0,0,0,0,0,0,0,0,0,0,0,0,0,0,0,0,0,0,0,0,0,0,0,0,0],FALSE];

ENDMODULE

--- Controller Data/v2600-510970_CAADRIA/RAPID/TASK4/SYSMOD/RRC_UserInteraction.sys ---
MODULE RRC_UserInteraction (SYSMODULE, NOSTEPIN)
    !***********************************************************************************
    !
    ! ETH Zurich / Robotic Fabrication Lab
    ! HIB C 13 / Stefano-Franscini-Platz 1
    ! CH-8093 Zurich
    !
    !***********************************************************************************
    !
    ! PROJECT     :  RRC - Rapid Robot Communication
    !
    ! FUNCTION    :  General Utilities Library
    !
    ! AUTHOR      :  Philippe Fleischmann
    !
    ! EMAIL       :  rrc@arch.ethz.ch
    !
    ! HISTORY     :  2019.02.22
    !
    ! Copyright   :  ETH Zurich (CH) 2019
    !                - Philippe Fleischmann
    !                - Michael Lyrenmann
    !                - Gonzalo Casas
    !
    ! License     :  This code base is governed by an EULA (End-User License Agreement)
    !                which you have received together with the software.
    !                You are not allowed to use the software on a real robots
    !                without a signed EULA.
    !
    !                A copy of the EULA content is in the controller task (T_CTRL).
    !
    !***********************************************************************************

    !************************************************
    ! Function    :     Teach Pendant (old FelxPendant) Message
    ! Programmer  :     Philippe Fleischmann
    ! Date        :     2019.02.22
    !***************** ETH Zurich *******************
    !
    PROC r_RRC_TPMsg(string stMsg)
        !
        ! Clear Msg Panel
        TPErase;
        !
        ! Msg for user
        TPWrite stMsg;
        !
        ! Time to read the Msg
        WaitTime n_RRC_TimeTPMsg;
        RETURN ;
    ERROR
        ! Placeholder for Error Code...
    ENDPROC

    !************************************************
    ! Function    :     Teach Pendant (old FelxPendant) Error Message
    ! Programmer  :     Philippe Fleischmann
    ! Date        :     2019.02.22
    !***************** ETH Zurich *******************
    !
    PROC r_RRC_TPErrMsg(num nErrno\switch StopTask\switch StopAllTasks)
        !
        ! Clear Msg Panel
        TPErase;
        !
        ! Write error number
        TPWrite "ERRNO = "\Num:=nErrno;
        !
        ! Stop task
        IF Present(StopTask) Stop;
        !
        ! Stop all normal tasks
        IF Present(StopAllTasks) Stop\AllMoveTasks;
        RETURN ;
    ERROR
        ! Placeholder for Error Code...
    ENDPROC

    !************************************************
    ! Function    :     Event Log Message
    ! Programmer  :     Philippe Fleischmann
    ! Date        :     2019.02.22
    !***************** ETH Zurich *******************
    !
    PROC r_RRC_EvLogMsg(string stHeader,string stMsg)
        !
        ! Msg for user
        ErrWrite\I,stHeader+" "+stMsg,"rLogMsg";
        RETURN ;
    ERROR
        ! Placeholder for Error Code...
    ENDPROC

    !************************************************
    ! Function    :     User interface message
    ! Programmer  :     Philippe Fleischmann
    ! Date        :     2019.02.22
    !***************** ETH Zurich *******************
    !
    FUNC string f_RRC_UIMsg(string stMsgHeader,string stMsgL1,\string stMsgL2,\string stMsgL3,\string stMsgL4,\string stMsgL5,string stBtn1\string stBtn2\string stBtn3\string stBtn4\string stBtn5,icondata icIcon)
        VAR num nAnswer;
        VAR string stMsg{5};
        VAR string stBtn{5};
        VAR string stAnswer;
        !
        ! Initialize variables
        stMsg:=["","","","",""];
        stBtn:=["","","","",""];
        !
        ! Load meassge
        stMsg{1}:=stMsgL1;
        IF Present(stMsgL2) stMsg{2}:=stMsgL2;
        IF Present(stMsgL3) stMsg{3}:=stMsgL3;
        IF Present(stMsgL4) stMsg{4}:=stMsgL4;
        IF Present(stMsgL5) stMsg{5}:=stMsgL5;
        !
        ! Load buttons
        stBtn{1}:=stBtn1;
        IF Present(stBtn2) stBtn{2}:=stBtn2;
        IF Present(stBtn3) stBtn{3}:=stBtn3;
        IF Present(stBtn4) stBtn{4}:=stBtn4;
        IF Present(stBtn5) stBtn{5}:=stBtn5;
        !
        ! Msg for user
        nAnswer:=UIMessageBox(
            \Header:=stMsgHeader
            \MsgArray:=stMsg
            \BtnArray:=stBtn
            \Icon:=icIcon);
        !
        ! handle user answer
        IF nAnswer=1 stAnswer:=stBtn{1};
        IF nAnswer=2 stAnswer:=stBtn{2};
        IF nAnswer=3 stAnswer:=stBtn{3};
        IF nAnswer=4 stAnswer:=stBtn{4};
        IF nAnswer=5 stAnswer:=stBtn{5};
        !
        ! Return user answer as string
        RETURN stAnswer;
    ERROR
        ! Placeholder for Error Code...
    ENDFUNC

    !************************************************
    ! Function    :     User interface numerical entry
    ! Programmer  :     Philippe Fleischmann
    ! Date        :     2019.02.22
    !***************** ETH Zurich *******************
    !
    FUNC num f_RRC_UINumEntry(string stMsgHeader,string stMsgL1,\string stMsgL2,\string stMsgL3,\string stMsgL4,\string stMsgL5,num nMin,num nMax,\num nDefault,icondata icIcon)
        VAR string stMsg{5};
        VAR num nAnswer;
        VAR num nInitValue;
        !
        ! Initialize variables
        stMsg:=["","","","",""];
        nInitValue:=nMin;
        !
        ! Load meassge
        stMsg{1}:=stMsgL1;
        IF Present(stMsgL2) stMsg{2}:=stMsgL2;
        IF Present(stMsgL3) stMsg{3}:=stMsgL3;
        IF Present(stMsgL4) stMsg{4}:=stMsgL4;
        IF Present(stMsgL5) stMsg{5}:=stMsgL5;
        !
        ! Use default value when present
        IF Present(nDefault) nInitValue:=nDefault;
        !
        ! Msg for user
        nAnswer:=Round(UINumEntry(
            \Header:=stMsgHeader
            \MsgArray:=stMsg
            \Icon:=icIcon
            \InitValue:=nInitValue
            \MinValue:=nMin
            \MaxValue:=nMax)\Dec:=1);
        !
        ! Return user answer as string
        RETURN nAnswer;
    ERROR
        ! Placeholder for Error Code...
    ENDFUNC


ENDMODULE

--- Controller Data/v2600-510970_CAADRIA/HOME/blickfeld7/T_ROB1.mod ---
MODULE MainModule
VAR speeddata Work:= [100,20,5000,1000];
PERS tooldata custom_tool1 := [TRUE, [[-234.48,-412.72,208.37], [0.624338,0.331967,-0.624338,0.331967]], [18,[0.10,0.00,0.00],[1,0,0,0],0,0,0]];
PROC Main()
! 20260323_yaya_ABB_update widest printing bed.gh [T_ROB1]
! 24/03/2026 16:29:50
! Generated with TACO for ABB
! http://taco.blickfeld7.com
! =====================================
ConfL \Off;
ConfJ \Off;
MoveL [[1520.01,-24.73,-524.72],[0.032971,0.999448,0.003972,-0.00071],[0,-1,-1,0],[0,9E9,9E9,9E9,9E9,9E9]],Work,fine,custom_tool1\WObj:=WObj0;
MoveL [[1520.01,-24.73,-624.72],[0.032971,0.999448,0.003972,-0.00071],[0,-1,-1,0],[0,9E9,9E9,9E9,9E9,9E9]],Work,fine,custom_tool1\WObj:=WObj0;
WaitTime 1;
SetDo Local_IO_0_DO2,1;
WaitTime 1;
MoveL [[1520.01,-24.73,-624.72],[0.032971,0.999448,0.003972,-0.00071],[0,-1,-1,0],[0,9E9,9E9,9E9,9E9,9E9]],Work,z10,custom_tool1\WObj:=WObj0;
MoveL [[1520.18,-34.73,-624.73],[0.032971,0.999448,0.003972,-0.00071],[0,-1,-1,0],[0,9E9,9E9,9E9,9E9,9E9]],Work,z10,custom_tool1\WObj:=WObj0;
MoveL [[1520.34,-44.73,-624.74],[0.032971,0.999448,0.003972,-0.00071],[0,-1,-1,0],[0,9E9,9E9,9E9,9E9,9E9]],Work,z10,custom_tool1\WObj:=WObj0;
MoveL [[1520.51,-54.73,-624.76],[0.032971,0.999448,0.003972,-0.00071],[0,-1,-1,0],[0,9E9,9E9,9E9,9E9,9E9]],Work,z10,custom_tool1\WObj:=WObj0;
MoveL [[1520.67,-64.73,-624.77],[0.032971,0.999448,0.003972,-0.00071],[0,-1,-1,0],[0,9E9,9E9,9E9,9E9,9E9]],Work,z10,custom_tool1\WObj:=WObj0;
MoveL [[1520.84,-74.73,-624.79],[0.032971,0.999448,0.003972,-0.00071],[0,-1,-1,0],[0,9E9,9E9,9E9,9E9,9E9]],Work,z10,custom_tool1\WObj:=WObj0;
MoveL [[1521,-84.72,-624.8],[0.032971,0.999448,0.003972,-0.00071],[0,-1,-1,0],[0,9E9,9E9,9E9,9E9,9E9]],Work,z10,custom_tool1\WObj:=WObj0;
MoveL [[1521.17,-94.72,-624.81],[0.032971,0.999448,0.003972,-0.00071],[0,-1,-1,0],[0,9E9,9E9,9E9,9E9,9E9]],Work,z10,custom_tool1\WObj:=WObj0;
MoveL [[1521.33,-104.72,-624.83],[0.032971,0.999448,0.003972,-0.00071],[0,-1,-1,0],[0,9E9,9E9,9E9,9E9,9E9]],Work,z10,custom_tool1\WObj:=WObj0;
MoveL [[1521.5,-114.72,-624.84],[0.032971,0.999448,0.003972,-0.00071],[0,-1,-1,0],[0,9E9,9E9,9E9,9E9,9E9]],Work,z10,custom_tool1\WObj:=WObj0;
MoveL [[1521.66,-124.72,-624.86],[0.032971,0.999448,0.003972,-0.00071],[0,-1,-1,0],[0,9E9,9E9,9E9,9E9,9E9]],Work,z10,custom_tool1\WObj:=WObj0;
MoveL [[1512.75,-128.8,-624.84],[0.032971,0.999448,0.003972,-0.00071],[0,-1,-1,0],[0,9E9,9E9,9E9,9E9,9E9]],Work,z10,custom_tool1\WObj:=WObj0;
MoveL [[1505.52,-135.48,-624.84],[0.032971,0.999448,0.003972,-0.00071],[0,-1,-1,0],[0,9E9,9E9,9E9,9E9,9E9]],Work,z10,custom_tool1\WObj:=WObj0;
MoveL [[1500.73,-144.2,-624.84],[0.032971,0.999448,0.003972,-0.00071],[0,-1,-1,0],[0,9E9,9E9,9E9,9E9,9E9]],Work,z10,custom_tool1\WObj:=WObj0;
MoveL [[1499.12,-154.06,-624.85],[0.032971,0.999448,0.003972,-0.00071],[0,-1,-1,0],[0,9E9,9E9,9E9,9E9,9E9]],Work,z10,custom_tool1\WObj:=WObj0;
MoveL [[1499.27,-164.06,-624.87],[0.032971,0.999448,0.003972,-0.00071],[0,-1,-1,0],[0,9E9,9E9,9E9,9E9,9E9]],Work,z10,custom_tool1\WObj:=WObj0;
MoveL [[1499.44,-174.06,-624.88],[0.032971,0.999448,0.003972,-0.00071],[0,-1,-1,0],[0,9E9,9E9,9E9,9E9,9E9]],Work,z10,custom_tool1\WObj:=WObj0;
MoveL [[1499.6,-184.06,-624.89],[0.032971,0.999448,0.003972,-0.00071],[0,-1,-1,0],[0,9E9,9E9,9E9,9E9,9E9]],Work,z10,custom_tool1\WObj:=WObj0;
MoveL [[1499.77,-194.06,-624.91],[0.032971,0.999448,0.003972,-0.00071],[0,-1,-1,0],[0,9E9,9E9,9E9,9E9,9E9]],Work,z10,custom_tool1\WObj:=WObj0;
MoveL [[1499.93,-204.05,-624.92],[0.032971,0.999448,0.003972,-0.00071],[0,-1,-1,0],[0,9E9,9E9,9E9,9E9,9E9]],Work,z10,custom_tool1\WObj:=WObj0;
MoveL [[1500.1,-214.05,-624.93],[0.032971,0.999448,0.003972,-0.00071],[0,-1,-1,0],[0,9E9,9E9,9E9,9E9,9E9]],Work,z10,custom_tool1\WObj:=WObj0;
MoveL [[1500.26,-224.05,-624.95],[0.032971,0.999448,0.003972,-0.00071],[0,-1,-1,0],[0,9E9,9E9,9E9,9E9,9E9]],Work,z10,custom_tool1\WObj:=WObj0;
MoveL [[1500.42,-234.05,-624.96],[0.032971,0.999448,0.003972,-0.00071],[0,-1,-1,0],[0,9E9,9E9,9E9,9E9,9E9]],Work,z10,custom_tool1\WObj:=WObj0;
MoveL [[1500.59,-244.05,-624.98],[0.032971,0.999448,0.003972,-0.00071],[0,-1,-1,0],[0,9E9,9E9,9E9,9E9,9E9]],Work,z10,custom_tool1\WObj:=WObj0;
MoveL [[1500.75,-254.05,-624.99],[0.032971,0.999448,0.003972,-0.00071],[0,-1,-1,0],[0,9E9,9E9,9E9,9E9,9E9]],Work,z10,custom_tool1\WObj:=WObj0;
MoveL [[1500.92,-264.05,-625],[0.032971,0.999448,0.003972,-0.00071],[0,-1,-1,0],[0,9E9,9E9,9E9,9E9,9E9]],Work,z10,custom_tool1\WObj:=WObj0;
MoveL [[1501.08,-274.05,-625.02],[0.032971,0.999448,0.003972,-0.00071],[0,-1,-1,0],[0,9E9,9E9,9E9,9E9,9E9]],Work,z10,custom_tool1\WObj:=WObj0;
MoveL [[1501.25,-284.04,-625.03],[0.032971,0.999448,0.003972,-0.00071],[0,-1,-1,0],[0,9E9,9E9,9E9,9E9,9E9]],Work,z10,custom_tool1\WObj:=WObj0;
MoveL [[1501.41,-294.04,-625.05],[0.032971,0.999448,0.003972,-0.00071],[0,-1,-1,0],[0,9E9,9E9,9E9,9E9,9E9]],Work,z10,custom_tool1\WObj:=WObj0;
MoveL [[1501.58,-304.04,-625.06],[0.032971,0.999448,0.003972,-0.00071],[0,-1,-1,0],[0,9E9,9E9,9E9,9E9,9E9]],Work,z10,custom_tool1\WObj:=WObj0;
MoveL [[1501.74,-314.04,-625.07],[0.032971,0.999448,0.003972,-0.00071],[0,-1,-1,0],[0,9E9,9E9,9E9,9E9,9E9]],Work,z10,custom_tool1\WObj:=WObj0;
MoveL [[1501.91,-324.04,-625.09],[0.032971,0.999448,0.003972,-0.00071],[0,-1,-1,0],[0,9E9,9E9,9E9,9E9,9E9]],Work,z10,custom_tool1\WObj:=WObj0;
MoveL [[1502.07,-334.04,-625.1],[0.032971,0.999448,0.003972,-0.00071],[0,-1,-1,0],[0,9E9,9E9,9E9,9E9,9E9]],Work,z10,custom_tool1\WObj:=WObj0;
MoveL [[1502.24,-344.04,-625.12],[0.032971,0.999448,0.003972,-0.00071],[0,-1,-1,0],[0,9E9,9E9,9E9,9E9,9E9]],Work,z10,custom_tool1\WObj:=WObj0;
MoveL [[1502.4,-354.03,-625.13],[0.032971,0.999448,0.003972,-0.00071],[0,-1,-1,0],[0,9E9,9E9,9E9,9E9,9E9]],Work,z10,custom_tool1\WObj:=WObj0;
MoveL [[1502.57,-364.03,-625.14],[0.032971,0.999448,0.003972,-0.00071],[0,-1,-1,0],[0,9E9,9E9,9E9,9E9,9E9]],Work,z10,custom_tool1\WObj:=WObj0;
MoveL [[1502.73,-374.03,-625.16],[0.032971,0.999448,0.003972,-0.00071],[0,-1,-1,0],[0,9E9,9E9,9E9,9E9,9E9]],Work,z10,custom_tool1\WObj:=WObj0;
MoveL [[1503,-384.02,-625.17],[0.032971,0.999448,0.003972,-0.00071],[0,-1,-1,0],[0,9E9,9E9,9E9,9E9,9E9]],Work,z10,custom_tool1\WObj:=WObj0;
MoveL [[1505.08,-393.8,-625.19],[0.032971,0.999448,0.003972,-0.00071],[0,-1,-1,0],[0,9E9,9E9,9E9,9E9,9E9]],Work,z10,custom_tool1\WObj:=WObj0;
MoveL [[1510.34,-402.23,-625.21],[0.032971,0.999448,0.003972,-0.00071],[0,-1,-1,0],[0,9E9,9E9,9E9,9E9,9E9]],Work,z10,custom_tool1\WObj:=WObj0;
MoveL [[1517.95,-408.51,-625.23],[0.032971,0.999448,0.003972,-0.00071],[0,-1,-1,0],[0,9E9,9E9,9E9,9E9,9E9]],Work,z10,custom_tool1\WObj:=WObj0;
MoveL [[1527.08,-412.11,-625.26],[0.032971,0.999448,0.003972,-0.00071],[0,-1,-1,0],[0,9E9,9E9,9E9,9E9,9E9]],Work,z10,custom_tool1\WObj:=WObj0;
MoveL [[1537,-413.13,-625.28],[0.032971,0.999448,0.003972,-0.00071],[0,-1,-1,0],[0,9E9,9E9,9E9,9E9,9E9]],Work,z10,custom_tool1\WObj:=WObj0;
MoveL [[1547,-412.96,-625.3],[0.032971,0.999448,0.003972,-0.00071],[0,-1,-1,0],[0,9E9,9E9,9E9,9E9,9E9]],Work,z10,custom_tool1\WObj:=WObj0;
MoveL [[1557,-412.79,-625.32],[0.032971,0.999448,0.003972,-0.00071],[0,-1,-1,0],[0,9E9,9E9,9E9,9E9,9E9]],Work,z10,custom_tool1\WObj:=WObj0;
MoveL [[1567,-412.63,-625.34],[0.032971,0.999448,0.003972,-0.00071],[0,-1,-1,0],[0,9E9,9E9,9E9,9E9,9E9]],Work,z10,custom_tool1\WObj:=WObj0;
MoveL [[1577,-412.47,-625.36],[0.032971,0.999448,0.003972,-0.00071],[0,-1,-1,0],[0,9E9,9E9,9E9,9E9,9E9]],Work,z10,custom_tool1\WObj:=WObj0;
MoveL [[1586.99,-412.3,-625.38],[0.032971,0.999448,0.003972,-0.00071],[0,-1,-1,0],[0,9E9,9E9,9E9,9E9,9E9]],Work,z10,custom_tool1\WObj:=WObj0;
MoveL [[1596.97,-411.84,-625.4],[0.032971,0.999448,0.003972,-0.00071],[0,-1,-1,0],[0,9E9,9E9,9E9,9E9,9E9]],Work,z10,custom_tool1\WObj:=WObj0;
MoveL [[1606.72,-409.69,-625.41],[0.032971,0.999448,0.003972,-0.00071],[0,-1,-1,0],[0,9E9,9E9,9E9,9E9,9E9]],Work,z10,custom_tool1\WObj:=WObj0;
MoveL [[1614.94,-404,-625.42],[0.032971,0.999448,0.003972,-0.00071],[0,-1,-1,0],[0,9E9,9E9,9E9,9E9,9E9]],Work,z10,custom_tool1\WObj:=WObj0;
MoveL [[1620.85,-396.06,-625.42],[0.032971,0.999448,0.003972,-0.00071],[0,-1,-1,0],[0,9E9,9E9,9E9,9E9,9E9]],Work,z10,custom_tool1\WObj:=WObj0;
MoveL [[1624.01,-386.73,-625.42],[0.032971,0.999448,0.003972,-0.00071],[0,-1,-1,0],[0,9E9,9E9,9E9,9E9,9E9]],Work,z10,custom_tool1\WObj:=WObj0;
MoveL [[1624.79,-376.8,-625.4],[0.032971,0.999448,0.003972,-0.00071],[0,-1,-1,0],[0,9E9,9E9,9E9,9E9,9E9]],Work,z10,custom_tool1\WObj:=WObj0;
MoveL [[1624.63,-366.8,-625.39],[0.032971,0.999448,0.003972,-0.00071],[0,-1,-1,0],[0,9E9,9E9,9E9,9E9,9E9]],Work,z10,custom_tool1\WObj:=WObj0;
MoveL [[1624.46,-356.8,-625.38],[0.032971,0.999448,0.003972,-0.00071],[0,-1,-1,0],[0,9E9,9E9,9E9,9E9,9E9]],Work,z10,custom_tool1\WObj:=WObj0;
MoveL [[1624.3,-346.8,-625.36],[0.032971,0.999448,0.003972,-0.00071],[0,-1,-1,0],[0,9E9,9E9,9E9,9E9,9E9]],Work,z10,custom_tool1\WObj:=WObj0;
MoveL [[1624.14,-336.8,-625.35],[0.032971,0.999448,0.003972,-0.00071],[0,-1,-1,0],[0,9E9,9E9,9E9,9E9,9E9]],Work,z10,custom_tool1\WObj:=WObj0;
MoveL [[1623.97,-326.8,-625.33],[0.032971,0.999448,0.003972,-0.00071],[0,-1,-1,0],[0,9E9,9E9,9E9,9E9,9E9]],Work,z10,custom_tool1\WObj:=WObj0;
MoveL [[1623.81,-316.8,-625.32],[0.032971,0.999448,0.003972,-0.00071],[0,-1,-1,0],[0,9E9,9E9,9E9,9E9,9E9]],Work,z10,custom_tool1\WObj:=WObj0;
MoveL [[1623.64,-306.81,-625.31],[0.032971,0.999448,0.003972,-0.00071],[0,-1,-1,0],[0,9E9,9E9,9E9,9E9,9E9]],Work,z10,custom_tool1\WObj:=WObj0;
MoveL [[1623.48,-296.81,-625.29],[0.032971,0.999448,0.003972,-0.00071],[0,-1,-1,0],[0,9E9,9E9,9E9,9E9,9E9]],Work,z10,custom_tool1\WObj:=WObj0;
MoveL [[1623.31,-286.81,-625.28],[0.032971,0.999448,0.003972,-0.00071],[0,-1,-1,0],[0,9E9,9E9,9E9,9E9,9E9]],Work,z10,custom_tool1\WObj:=WObj0;
MoveL [[1623.15,-276.81,-625.27],[0.032971,0.999448,0.003972,-0.00071],[0,-1,-1,0],[0,9E9,9E9,9E9,9E9,9E9]],Work,z10,custom_tool1\WObj:=WObj0;
MoveL [[1622.98,-266.81,-625.25],[0.032971,0.999448,0.003972,-0.00071],[0,-1,-1,0],[0,9E9,9E9,9E9,9E9,9E9]],Work,z10,custom_tool1\WObj:=WObj0;
MoveL [[1622.82,-256.81,-625.24],[0.032971,0.999448,0.003972,-0.00071],[0,-1,-1,0],[0,9E9,9E9,9E9,9E9,9E9]],Work,z10,custom_tool1\WObj:=WObj0;
MoveL [[1622.65,-246.81,-625.22],[0.032971,0.999448,0.003972,-0.00071],[0,-1,-1,0],[0,9E9,9E9,9E9,9E9,9E9]],Work,z10,custom_tool1\WObj:=WObj0;
MoveL [[1622.49,-236.81,-625.21],[0.032971,0.999448,0.003972,-0.00071],[0,-1,-1,0],[0,9E9,9E9,9E9,9E9,9E9]],Work,z10,custom_tool1\WObj:=WObj0;
MoveL [[1622.32,-226.82,-625.2],[0.032971,0.999448,0.003972,-0.00071],[0,-1,-1,0],[0,9E9,9E9,9E9,9E9,9E9]],Work,z10,custom_tool1\WObj:=WObj0;
MoveL [[1622.16,-216.82,-625.18],[0.032971,0.999448,0.003972,-0.00071],[0,-1,-1,0],[0,9E9,9E9,9E9,9E9,9E9]],Work,z10,custom_tool1\WObj:=WObj0;
MoveL [[1621.99,-206.82,-625.17],[0.032971,0.999448,0.003972,-0.00071],[0,-1,-1,0],[0,9E9,9E9,9E9,9E9,9E9]],Work,z10,custom_tool1\WObj:=WObj0;
MoveL [[1621.83,-196.82,-625.15],[0.032971,0.999448,0.003972,-0.00071],[0,-1,-1,0],[0,9E9,9E9,9E9,9E9,9E9]],Work,z10,custom_tool1\WObj:=WObj0;
MoveL [[1621.66,-186.82,-625.14],[0.032971,0.999448,0.003972,-0.00071],[0,-1,-1,0],[0,9E9,9E9,9E9,9E9,9E9]],Work,z10,custom_tool1\WObj:=WObj0;
MoveL [[1621.5,-176.82,-625.13],[0.032971,0.999448,0.003972,-0.00071],[0,-1,-1,0],[0,9E9,9E9,9E9,9E9,9E9]],Work,z10,custom_tool1\WObj:=WObj0;
MoveL [[1621.33,-166.82,-625.11],[0.032971,0.999448,0.003972,-0.00071],[0,-1,-1,0],[0,9E9,9E9,9E9,9E9,9E9]],Work,z10,custom_tool1\WObj:=WObj0;
MoveL [[1621.17,-156.83,-625.1],[0.032971,0.999448,0.003972,-0.00071],[0,-1,-1,0],[0,9E9,9E9,9E9,9E9,9E9]],Work,z10,custom_tool1\WObj:=WObj0;
MoveL [[1620.06,-146.93,-625.08],[0.032971,0.999448,0.003972,-0.00071],[0,-1,-1,0],[0,9E9,9E9,9E9,9E9,9E9]],Work,z10,custom_tool1\WObj:=WObj0;
MoveL [[1616.76,-137.65,-625.06],[0.032971,0.999448,0.003972,-0.00071],[0,-1,-1,0],[0,9E9,9E9,9E9,9E9,9E9]],Work,z10,custom_tool1\WObj:=WObj0;
MoveL [[1610.67,-129.78,-625.04],[0.032971,0.999448,0.003972,-0.00071],[0,-1,-1,0],[0,9E9,9E9,9E9,9E9,9E9]],Work,z10,custom_tool1\WObj:=WObj0;
MoveL [[1602.22,-124.44,-625.02],[0.032971,0.999448,0.003972,-0.00071],[0,-1,-1,0],[0,9E9,9E9,9E9,9E9,9E9]],Work,z10,custom_tool1\WObj:=WObj0;
MoveL [[1592.43,-122.5,-624.99],[0.032971,0.999448,0.003972,-0.00071],[0,-1,-1,0],[0,9E9,9E9,9E9,9E9,9E9]],Work,z10,custom_tool1\WObj:=WObj0;
MoveL [[1582.45,-122.34,-624.97],[0.032971,0.999448,0.003972,-0.00071],[0,-1,-1,0],[0,9E9,9E9,9E9,9E9,9E9]],Work,z10,custom_tool1\WObj:=WObj0;
MoveL [[1572.45,-122.5,-624.95],[0.032971,0.999448,0.003972,-0.00071],[0,-1,-1,0],[0,9E9,9E9,9E9,9E9,9E9]],Work,z10,custom_tool1\WObj:=WObj0;
MoveL [[1562.45,-122.67,-624.93],[0.032971,0.999448,0.003972,-0.00071],[0,-1,-1,0],[0,9E9,9E9,9E9,9E9,9E9]],Work,z10,custom_tool1\WObj:=WObj0;
MoveL [[1552.45,-122.83,-624.92],[0.032971,0.999448,0.003972,-0.00071],[0,-1,-1,0],[0,9E9,9E9,9E9,9E9,9E9]],Work,z10,custom_tool1\WObj:=WObj0;
MoveL [[1542.45,-123,-624.9],[0.032971,0.999448,0.003972,-0.00071],[0,-1,-1,0],[0,9E9,9E9,9E9,9E9,9E9]],Work,z10,custom_tool1\WObj:=WObj0;
MoveL [[1532.45,-123.16,-624.88],[0.032971,0.999448,0.003972,-0.00071],[0,-1,-1,0],[0,9E9,9E9,9E9,9E9,9E9]],Work,z10,custom_tool1\WObj:=WObj0;
MoveL [[1522.58,-124.52,-624.86],[0.032971,0.999448,0.003972,-0.00071],[0,-1,-1,0],[0,9E9,9E9,9E9,9E9,9E9]],Work,z10,custom_tool1\WObj:=WObj0;
MoveL [[1531.38,-124.77,-624.88],[0.032971,0.999448,0.003972,-0.00071],[0,-1,-1,0],[0,9E9,9E9,9E9,9E9,9E9]],Work,z10,custom_tool1\WObj:=WObj0;
MoveL [[1540.19,-125.03,-624.89],[0.032971,0.999448,0.003972,-0.00071],[0,-1,-1,0],[0,9E9,9E9,9E9,9E9,9E9]],Work,z10,custom_tool1\WObj:=WObj0;
MoveL [[1530.41,-127.16,-624.88],[0.032971,0.999448,0.003972,-0.00071],[0,-1,-1,0],[0,9E9,9E9,9E9,9E9,9E9]],Work,z10,custom_tool1\WObj:=WObj0;
MoveL [[1520.64,-129.28,-624.86],[0.032971,0.999448,0.003972,-0.00071],[0,-1,-1,0],[0,9E9,9E9,9E9,9E9,9E9]],Work,z10,custom_tool1\WObj:=WObj0;
MoveL [[1507.39,-136.25,-624.84],[0.032971,0.999448,0.003972,-0.00071],[0,-1,-1,0],[0,9E9,9E9,9E9,9E9,9E9]],Work,z10,custom_tool1\WObj:=WObj0;
MoveL [[1517.17,-134.13,-624.86],[0.032971,0.999448,0.003972,-0.00071],[0,-1,-1,0],[0,9E9,9E9,9E9,9E9,9E9]],Work,z10,custom_tool1\WObj:=WObj0;
MoveL [[1526.94,-132,-624.88],[0.032971,0.999448,0.003972,-0.00071],[0,-1,-1,0],[0,9E9,9E9,9E9,9E9,9E9]],Work,z10,custom_tool1\WObj:=WObj0;
MoveL [[1536.71,-129.88,-624.89],[0.032971,0.999448,0.003972,-0.00071],[0,-1,-1,0],[0,9E9,9E9,9E9,9E9,9E9]],Work,z10,custom_tool1\WObj:=WObj0;
MoveL [[1546.48,-127.76,-624.91],[0.032971,0.999448,0.003972,-0.00071],[0,-1,-1,0],[0,9E9,9E9,9E9,9E9,9E9]],Work,z10,custom_tool1\WObj:=WObj0;
MoveL [[1556.25,-125.64,-624.93],[0.032971,0.999448,0.003972,-0.00071],[0,-1,-1,0],[0,9E9,9E9,9E9,9E9,9E9]],Work,z10,custom_tool1\WObj:=WObj0;
MoveL [[1568.61,-125,-624.95],[0.032971,0.999448,0.003972,-0.00071],[0,-1,-1,0],[0,9E9,9E9,9E9,9E9,9E9]],Work,z10,custom_tool1\WObj:=WObj0;
MoveL [[1580.97,-124.36,-624.97],[0.032971,0.999448,0.003972,-0.00071],[0,-1,-1,0],[0,9E9,9E9,9E9,9E9,9E9]],Work,z10,custom_tool1\WObj:=WObj0;
MoveL [[1571.2,-126.48,-624.96],[0.032971,0.999448,0.003972,-0.00071],[0,-1,-1,0],[0,9E9,9E9,9E9,9E9,9E9]],Work,z10,custom_tool1\WObj:=WObj0;
MoveL [[1561.43,-128.61,-624.94],[0.032971,0.999448,0.003972,-0.00071],[0,-1,-1,0],[0,9E9,9E9,9E9,9E9,9E9]],Work,z10,custom_tool1\WObj:=WObj0;
MoveL [[1551.66,-130.73,-624.92],[0.032971,0.999448,0.003972,-0.00071],[0,-1,-1,0],[0,9E9,9E9,9E9,9E9,9E9]],Work,z10,custom_tool1\WObj:=WObj0;
MoveL [[1541.88,-132.85,-624.91],[0.032971,0.999448,0.003972,-0.00071],[0,-1,-1,0],[0,9E9,9E9,9E9,9E9,9E9]],Work,z10,custom_tool1\WObj:=WObj0;
MoveL [[1532.11,-134.97,-624.89],[0.032971,0.999448,0.003972,-0.00071],[0,-1,-1,0],[0,9E9,9E9,9E9,9E9,9E9]],Work,z10,custom_tool1\WObj:=WObj0;
MoveL [[1522.34,-137.1,-624.87],[0.032971,0.999448,0.003972,-0.00071],[0,-1,-1,0],[0,9E9,9E9,9E9,9E9,9E9]],Work,z10,custom_tool1\WObj:=WObj0;
MoveL [[1512.57,-139.22,-624.86],[0.032971,0.999448,0.003972,-0.00071],[0,-1,-1,0],[0,9E9,9E9,9E9,9E9,9E9]],Work,z10,custom_tool1\WObj:=WObj0;
MoveL [[1502.5,-145.5,-624.85],[0.032971,0.999448,0.003972,-0.00071],[0,-1,-1,0],[0,9E9,9E9,9E9,9E9,9E9]],Work,z10,custom_tool1\WObj:=WObj0;
MoveL [[1512.28,-143.37,-624.86],[0.032971,0.999448,0.003972,-0.00071],[0,-1,-1,0],[0,9E9,9E9,9E9,9E9,9E9]],Work,z10,custom_tool1\WObj:=WObj0;
MoveL [[1522.05,-141.25,-624.88],[0.032971,0.999448,0.003972,-0.00071],[0,-1,-1,0],[0,9E9,9E9,9E9,9E9,9E9]],Work,z10,custom_tool1\WObj:=WObj0;
MoveL [[1531.82,-139.13,-624.9],[0.032971,0.999448,0.003972,-0.00071],[0,-1,-1,0],[0,9E9,9E9,9E9,9E9,9E9]],Work,z10,custom_tool1\WObj:=WObj0;
MoveL [[1541.59,-137.01,-624.91],[0.032971,0.999448,0.003972,-0.00071],[0,-1,-1,0],[0,9E9,9E9,9E9,9E9,9E9]],Work,z10,custom_tool1\WObj:=WObj0;
MoveL [[1551.37,-134.88,-624.93],[0.032971,0.999448,0.003972,-0.00071],[0,-1,-1,0],[0,9E9,9E9,9E9,9E9,9E9]],Work,z10,custom_tool1\WObj:=WObj0;
MoveL [[1561.14,-132.76,-624.95],[0.032971,0.999448,0.003972,-0.00071],[0,-1,-1,0],[0,9E9,9E9,9E9,9E9,9E9]],Work,z10,custom_tool1\WObj:=WObj0;
MoveL [[1570.91,-130.64,-624.96],[0.032971,0.999448,0.003972,-0.00071],[0,-1,-1,0],[0,9E9,9E9,9E9,9E9,9E9]],Work,z10,custom_tool1\WObj:=WObj0;
MoveL [[1580.68,-128.52,-624.98],[0.032971,0.999448,0.003972,-0.00071],[0,-1,-1,0],[0,9E9,9E9,9E9,9E9,9E9]],Work,z10,custom_tool1\WObj:=WObj0;
MoveL [[1590.45,-126.39,-625],[0.032971,0.999448,0.003972,-0.00071],[0,-1,-1,0],[0,9E9,9E9,9E9,9E9,9E9]],Work,z10,custom_tool1\WObj:=WObj0;
MoveL [[1603.48,-127.66,-625.02],[0.032971,0.999448,0.003972,-0.00071],[0,-1,-1,0],[0,9E9,9E9,9E9,9E9,9E9]],Work,z10,custom_tool1\WObj:=WObj0;
MoveL [[1593.71,-129.78,-625.01],[0.032971,0.999448,0.003972,-0.00071],[0,-1,-1,0],[0,9E9,9E9,9E9,9E9,9E9]],Work,z10,custom_tool1\WObj:=WObj0;
MoveL [[1583.94,-131.9,-624.99],[0.032971,0.999448,0.003972,-0.00071],[0,-1,-1,0],[0,9E9,9E9,9E9,9E9,9E9]],Work,z10,custom_tool1\WObj:=WObj0;
MoveL [[1574.16,-134.03,-624.97],[0.032971,0.999448,0.003972,-0.00071],[0,-1,-1,0],[0,9E9,9E9,9E9,9E9,9E9]],Work,z10,custom_tool1\WObj:=WObj0;
MoveL [[1564.39,-136.15,-624.96],[0.032971,0.999448,0.003972,-0.00071],[0,-1,-1,0],[0,9E9,9E9,9E9,9E9,9E9]],Work,z10,custom_tool1\WObj:=WObj0;
MoveL [[1554.62,-138.27,-624.94],[0.032971,0.999448,0.003972,-0.00071],[0,-1,-1,0],[0,9E9,9E9,9E9,9E9,9E9]],Work,z10,custom_tool1\WObj:=WObj0;
MoveL [[1544.85,-140.39,-624.92],[0.032971,0.999448,0.003972,-0.00071],[0,-1,-1,0],[0,9E9,9E9,9E9,9E9,9E9]],Work,z10,custom_tool1\WObj:=WObj0;
MoveL [[1535.08,-142.52,-624.91],[0.032971,0.999448,0.003972,-0.00071],[0,-1,-1,0],[0,9E9,9E9,9E9,9E9,9E9]],Work,z10,custom_tool1\WObj:=WObj0;
MoveL [[1525.3,-144.64,-624.89],[0.032971,0.999448,0.003972,-0.00071],[0,-1,-1,0],[0,9E9,9E9,9E9,9E9,9E9]],Work,z10,custom_tool1\WObj:=WObj0;
MoveL [[1515.53,-146.76,-624.87],[0.032971,0.999448,0.003972,-0.00071],[0,-1,-1,0],[0,9E9,9E9,9E9,9E9,9E9]],Work,z10,custom_tool1\WObj:=WObj0;
MoveL [[1505.76,-148.88,-624.86],[0.032971,0.999448,0.003972,-0.00071],[0,-1,-1,0],[0,9E9,9E9,9E9,9E9,9E9]],Work,z10,custom_tool1\WObj:=WObj0;
MoveL [[1501.14,-153.98,-624.86],[0.032971,0.999448,0.003972,-0.00071],[0,-1,-1,0],[0,9E9,9E9,9E9,9E9,9E9]],Work,z10,custom_tool1\WObj:=WObj0;
MoveL [[1510.91,-151.86,-624.87],[0.032971,0.999448,0.003972,-0.00071],[0,-1,-1,0],[0,9E9,9E9,9E9,9E9,9E9]],Work,z10,custom_tool1\WObj:=WObj0;
MoveL [[1520.68,-149.74,-624.89],[0.032971,0.999448,0.003972,-0.00071],[0,-1,-1,0],[0,9E9,9E9,9E9,9E9,9E9]],Work,z10,custom_tool1\WObj:=WObj0;
MoveL [[1530.45,-147.61,-624.9],[0.032971,0.999448,0.003972,-0.00071],[0,-1,-1,0],[0,9E9,9E9,9E9,9E9,9E9]],Work,z10,custom_tool1\WObj:=WObj0;
MoveL [[1540.23,-145.49,-624.92],[0.032971,0.999448,0.003972,-0.00071],[0,-1,-1,0],[0,9E9,9E9,9E9,9E9,9E9]],Work,z10,custom_tool1\WObj:=WObj0;
MoveL [[1550,-143.37,-624.94],[0.032971,0.999448,0.003972,-0.00071],[0,-1,-1,0],[0,9E9,9E9,9E9,9E9,9E9]],Work,z10,custom_tool1\WObj:=WObj0;
MoveL [[1559.77,-141.25,-624.95],[0.032971,0.999448,0.003972,-0.00071],[0,-1,-1,0],[0,9E9,9E9,9E9,9E9,9E9]],Work,z10,custom_tool1\WObj:=WObj0;
MoveL [[1569.54,-139.12,-624.97],[0.032971,0.999448,0.003972,-0.00071],[0,-1,-1,0],[0,9E9,9E9,9E9,9E9,9E9]],Work,z10,custom_tool1\WObj:=WObj0;
MoveL [[1579.31,-137,-624.99],[0.032971,0.999448,0.003972,-0.00071],[0,-1,-1,0],[0,9E9,9E9,9E9,9E9,9E9]],Work,z10,custom_tool1\WObj:=WObj0;
MoveL [[1589.09,-134.88,-625],[0.032971,0.999448,0.003972,-0.00071],[0,-1,-1,0],[0,9E9,9E9,9E9,9E9,9E9]],Work,z10,custom_tool1\WObj:=WObj0;
MoveL [[1598.86,-132.76,-625.02],[0.032971,0.999448,0.003972,-0.00071],[0,-1,-1,0],[0,9E9,9E9,9E9,9E9,9E9]],Work,z10,custom_tool1\WObj:=WObj0;
MoveL [[1611.82,-134.03,-625.05],[0.032971,0.999448,0.003972,-0.00071],[0,-1,-1,0],[0,9E9,9E9,9E9,9E9,9E9]],Work,z10,custom_tool1\WObj:=WObj0;
MoveL [[1602.05,-136.16,-625.03],[0.032971,0.999448,0.003972,-0.00071],[0,-1,-1,0],[0,9E9,9E9,9E9,9E9,9E9]],Work,z10,custom_tool1\WObj:=WObj0;
MoveL [[1592.28,-138.28,-625.02],[0.032971,0.999448,0.003972,-0.00071],[0,-1,-1,0],[0,9E9,9E9,9E9,9E9,9E9]],Work,z10,custom_tool1\WObj:=WObj0;
MoveL [[1582.51,-140.4,-625],[0.032971,0.999448,0.003972,-0.00071],[0,-1,-1,0],[0,9E9,9E9,9E9,9E9,9E9]],Work,z10,custom_tool1\WObj:=WObj0;
MoveL [[1572.73,-142.52,-624.98],[0.032971,0.999448,0.003972,-0.00071],[0,-1,-1,0],[0,9E9,9E9,9E9,9E9,9E9]],Work,z10,custom_tool1\WObj:=WObj0;
MoveL [[1562.96,-144.65,-624.97],[0.032971,0.999448,0.003972,-0.00071],[0,-1,-1,0],[0,9E9,9E9,9E9,9E9,9E9]],Work,z10,custom_tool1\WObj:=WObj0;
MoveL [[1553.19,-146.77,-624.95],[0.032971,0.999448,0.003972,-0.00071],[0,-1,-1,0],[0,9E9,9E9,9E9,9E9,9E9]],Work,z10,custom_tool1\WObj:=WObj0;
MoveL [[1543.42,-148.89,-624.93],[0.032971,0.999448,0.003972,-0.00071],[0,-1,-1,0],[0,9E9,9E9,9E9,9E9,9E9]],Work,z10,custom_tool1\WObj:=WObj0;
MoveL [[1533.64,-151.01,-624.92],[0.032971,0.999448,0.003972,-0.00071],[0,-1,-1,0],[0,9E9,9E9,9E9,9E9,9E9]],Work,z10,custom_tool1\WObj:=WObj0;
MoveL [[1523.87,-153.14,-624.9],[0.032971,0.999448,0.003972,-0.00071],[0,-1,-1,0],[0,9E9,9E9,9E9,9E9,9E9]],Work,z10,custom_tool1\WObj:=WObj0;
MoveL [[1514.1,-155.26,-624.88],[0.032971,0.999448,0.003972,-0.00071],[0,-1,-1,0],[0,9E9,9E9,9E9,9E9,9E9]],Work,z10,custom_tool1\WObj:=WObj0;
MoveL [[1504.33,-157.38,-624.87],[0.032971,0.999448,0.003972,-0.00071],[0,-1,-1,0],[0,9E9,9E9,9E9,9E9,9E9]],Work,z10,custom_tool1\WObj:=WObj0;
MoveL [[1501.24,-162.15,-624.87],[0.032971,0.999448,0.003972,-0.00071],[0,-1,-1,0],[0,9E9,9E9,9E9,9E9,9E9]],Work,z10,custom_tool1\WObj:=WObj0;
MoveL [[1511.01,-160.02,-624.88],[0.032971,0.999448,0.003972,-0.00071],[0,-1,-1,0],[0,9E9,9E9,9E9,9E9,9E9]],Work,z10,custom_tool1\WObj:=WObj0;
MoveL [[1520.78,-157.9,-624.9],[0.032971,0.999448,0.003972,-0.00071],[0,-1,-1,0],[0,9E9,9E9,9E9,9E9,9E9]],Work,z10,custom_tool1\WObj:=WObj0;
MoveL [[1530.56,-155.78,-624.92],[0.032971,0.999448,0.003972,-0.00071],[0,-1,-1,0],[0,9E9,9E9,9E9,9E9,9E9]],Work,z10,custom_tool1\WObj:=WObj0;
MoveL [[1540.33,-153.66,-624.93],[0.032971,0.999448,0.003972,-0.00071],[0,-1,-1,0],[0,9E9,9E9,9E9,9E9,9E9]],Work,z10,custom_tool1\WObj:=WObj0;
MoveL [[1550.1,-151.53,-624.95],[0.032971,0.999448,0.003972,-0.00071],[0,-1,-1,0],[0,9E9,9E9,9E9,9E9,9E9]],Work,z10,custom_tool1\WObj:=WObj0;
MoveL [[1559.87,-149.41,-624.97],[0.032971,0.999448,0.003972,-0.00071],[0,-1,-1,0],[0,9E9,9E9,9E9,9E9,9E9]],Work,z10,custom_tool1\WObj:=WObj0;
MoveL [[1569.64,-147.29,-624.98],[0.032971,0.999448,0.003972,-0.00071],[0,-1,-1,0],[0,9E9,9E9,9E9,9E9,9E9]],Work,z10,custom_tool1\WObj:=WObj0;
MoveL [[1579.42,-145.16,-625],[0.032971,0.999448,0.003972,-0.00071],[0,-1,-1,0],[0,9E9,9E9,9E9,9E9,9E9]],Work,z10,custom_tool1\WObj:=WObj0;
MoveL [[1589.19,-143.04,-625.02],[0.032971,0.999448,0.003972,-0.00071],[0,-1,-1,0],[0,9E9,9E9,9E9,9E9,9E9]],Work,z10,custom_tool1\WObj:=WObj0;
MoveL [[1598.96,-140.92,-625.03],[0.032971,0.999448,0.003972,-0.00071],[0,-1,-1,0],[0,9E9,9E9,9E9,9E9,9E9]],Work,z10,custom_tool1\WObj:=WObj0;
MoveL [[1608.73,-138.8,-625.05],[0.032971,0.999448,0.003972,-0.00071],[0,-1,-1,0],[0,9E9,9E9,9E9,9E9,9E9]],Work,z10,custom_tool1\WObj:=WObj0;
MoveL [[1616.69,-141.16,-625.07],[0.032971,0.999448,0.003972,-0.00071],[0,-1,-1,0],[0,9E9,9E9,9E9,9E9,9E9]],Work,z10,custom_tool1\WObj:=WObj0;
MoveL [[1606.92,-143.29,-625.05],[0.032971,0.999448,0.003972,-0.00071],[0,-1,-1,0],[0,9E9,9E9,9E9,9E9,9E9]],Work,z10,custom_tool1\WObj:=WObj0;
MoveL [[1597.14,-145.41,-625.03],[0.032971,0.999448,0.003972,-0.00071],[0,-1,-1,0],[0,9E9,9E9,9E9,9E9,9E9]],Work,z10,custom_tool1\WObj:=WObj0;
MoveL [[1587.37,-147.53,-625.02],[0.032971,0.999448,0.003972,-0.00071],[0,-1,-1,0],[0,9E9,9E9,9E9,9E9,9E9]],Work,z10,custom_tool1\WObj:=WObj0;
MoveL [[1577.6,-149.65,-625],[0.032971,0.999448,0.003972,-0.00071],[0,-1,-1,0],[0,9E9,9E9,9E9,9E9,9E9]],Work,z10,custom_tool1\WObj:=WObj0;
MoveL [[1567.83,-151.78,-624.98],[0.032971,0.999448,0.003972,-0.00071],[0,-1,-1,0],[0,9E9,9E9,9E9,9E9,9E9]],Work,z10,custom_tool1\WObj:=WObj0;
MoveL [[1558.06,-153.9,-624.97],[0.032971,0.999448,0.003972,-0.00071],[0,-1,-1,0],[0,9E9,9E9,9E9,9E9,9E9]],Work,z10,custom_tool1\WObj:=WObj0;
MoveL [[1548.28,-156.02,-624.95],[0.032971,0.999448,0.003972,-0.00071],[0,-1,-1,0],[0,9E9,9E9,9E9,9E9,9E9]],Work,z10,custom_tool1\WObj:=WObj0;
MoveL [[1538.51,-158.14,-624.94],[0.032971,0.999448,0.003972,-0.00071],[0,-1,-1,0],[0,9E9,9E9,9E9,9E9,9E9]],Work,z10,custom_tool1\WObj:=WObj0;
MoveL [[1528.74,-160.27,-624.92],[0.032971,0.999448,0.003972,-0.00071],[0,-1,-1,0],[0,9E9,9E9,9E9,9E9,9E9]],Work,z10,custom_tool1\WObj:=WObj0;
MoveL [[1518.97,-162.39,-624.9],[0.032971,0.999448,0.003972,-0.00071],[0,-1,-1,0],[0,9E9,9E9,9E9,9E9,9E9]],Work,z10,custom_tool1\WObj:=WObj0;
MoveL [[1509.19,-164.51,-624.89],[0.032971,0.999448,0.003972,-0.00071],[0,-1,-1,0],[0,9E9,9E9,9E9,9E9,9E9]],Work,z10,custom_tool1\WObj:=WObj0;
MoveL [[1501.37,-170.3,-624.88],[0.032971,0.999448,0.003972,-0.00071],[0,-1,-1,0],[0,9E9,9E9,9E9,9E9,9E9]],Work,z10,custom_tool1\WObj:=WObj0;
MoveL [[1511.15,-168.18,-624.89],[0.032971,0.999448,0.003972,-0.00071],[0,-1,-1,0],[0,9E9,9E9,9E9,9E9,9E9]],Work,z10,custom_tool1\WObj:=WObj0;
MoveL [[1520.92,-166.06,-624.91],[0.032971,0.999448,0.003972,-0.00071],[0,-1,-1,0],[0,9E9,9E9,9E9,9E9,9E9]],Work,z10,custom_tool1\WObj:=WObj0;
MoveL [[1530.69,-163.93,-624.93],[0.032971,0.999448,0.003972,-0.00071],[0,-1,-1,0],[0,9E9,9E9,9E9,9E9,9E9]],Work,z10,custom_tool1\WObj:=WObj0;
MoveL [[1540.46,-161.81,-624.94],[0.032971,0.999448,0.003972,-0.00071],[0,-1,-1,0],[0,9E9,9E9,9E9,9E9,9E9]],Work,z10,custom_tool1\WObj:=WObj0;
MoveL [[1550.23,-159.69,-624.96],[0.032971,0.999448,0.003972,-0.00071],[0,-1,-1,0],[0,9E9,9E9,9E9,9E9,9E9]],Work,z10,custom_tool1\WObj:=WObj0;
MoveL [[1560.01,-157.57,-624.98],[0.032971,0.999448,0.003972,-0.00071],[0,-1,-1,0],[0,9E9,9E9,9E9,9E9,9E9]],Work,z10,custom_tool1\WObj:=WObj0;
MoveL [[1569.78,-155.44,-624.99],[0.032971,0.999448,0.003972,-0.00071],[0,-1,-1,0],[0,9E9,9E9,9E9,9E9,9E9]],Work,z10,custom_tool1\WObj:=WObj0;
MoveL [[1579.55,-153.32,-625.01],[0.032971,0.999448,0.003972,-0.00071],[0,-1,-1,0],[0,9E9,9E9,9E9,9E9,9E9]],Work,z10,custom_tool1\WObj:=WObj0;
MoveL [[1589.32,-151.2,-625.03],[0.032971,0.999448,0.003972,-0.00071],[0,-1,-1,0],[0,9E9,9E9,9E9,9E9,9E9]],Work,z10,custom_tool1\WObj:=WObj0;
MoveL [[1599.1,-149.08,-625.04],[0.032971,0.999448,0.003972,-0.00071],[0,-1,-1,0],[0,9E9,9E9,9E9,9E9,9E9]],Work,z10,custom_tool1\WObj:=WObj0;
MoveL [[1608.87,-146.95,-625.06],[0.032971,0.999448,0.003972,-0.00071],[0,-1,-1,0],[0,9E9,9E9,9E9,9E9,9E9]],Work,z10,custom_tool1\WObj:=WObj0;
MoveL [[1618.45,-148.97,-625.08],[0.032971,0.999448,0.003972,-0.00071],[0,-1,-1,0],[0,9E9,9E9,9E9,9E9,9E9]],Work,z10,custom_tool1\WObj:=WObj0;
MoveL [[1608.68,-151.09,-625.07],[0.032971,0.999448,0.003972,-0.00071],[0,-1,-1,0],[0,9E9,9E9,9E9,9E9,9E9]],Work,z10,custom_tool1\WObj:=WObj0;
MoveL [[1598.91,-153.21,-625.05],[0.032971,0.999448,0.003972,-0.00071],[0,-1,-1,0],[0,9E9,9E9,9E9,9E9,9E9]],Work,z10,custom_tool1\WObj:=WObj0;
MoveL [[1589.14,-155.33,-625.03],[0.032971,0.999448,0.003972,-0.00071],[0,-1,-1,0],[0,9E9,9E9,9E9,9E9,9E9]],Work,z10,custom_tool1\WObj:=WObj0;
MoveL [[1579.37,-157.46,-625.02],[0.032971,0.999448,0.003972,-0.00071],[0,-1,-1,0],[0,9E9,9E9,9E9,9E9,9E9]],Work,z10,custom_tool1\WObj:=WObj0;
MoveL [[1569.59,-159.58,-625],[0.032971,0.999448,0.003972,-0.00071],[0,-1,-1,0],[0,9E9,9E9,9E9,9E9,9E9]],Work,z10,custom_tool1\WObj:=WObj0;
MoveL [[1559.82,-161.7,-624.98],[0.032971,0.999448,0.003972,-0.00071],[0,-1,-1,0],[0,9E9,9E9,9E9,9E9,9E9]],Work,z10,custom_tool1\WObj:=WObj0;
MoveL [[1550.05,-163.82,-624.97],[0.032971,0.999448,0.003972,-0.00071],[0,-1,-1,0],[0,9E9,9E9,9E9,9E9,9E9]],Work,z10,custom_tool1\WObj:=WObj0;
MoveL [[1540.28,-165.95,-624.95],[0.032971,0.999448,0.003972,-0.00071],[0,-1,-1,0],[0,9E9,9E9,9E9,9E9,9E9]],Work,z10,custom_tool1\WObj:=WObj0;
MoveL [[1530.51,-168.07,-624.93],[0.032971,0.999448,0.003972,-0.00071],[0,-1,-1,0],[0,9E9,9E9,9E9,9E9,9E9]],Work,z10,custom_tool1\WObj:=WObj0;
MoveL [[1520.73,-170.19,-624.92],[0.032971,0.999448,0.003972,-0.00071],[0,-1,-1,0],[0,9E9,9E9,9E9,9E9,9E9]],Work,z10,custom_tool1\WObj:=WObj0;
MoveL [[1510.96,-172.31,-624.9],[0.032971,0.999448,0.003972,-0.00071],[0,-1,-1,0],[0,9E9,9E9,9E9,9E9,9E9]],Work,z10,custom_tool1\WObj:=WObj0;
MoveL [[1501.51,-178.46,-624.89],[0.032971,0.999448,0.003972,-0.00071],[0,-1,-1,0],[0,9E9,9E9,9E9,9E9,9E9]],Work,z10,custom_tool1\WObj:=WObj0;
MoveL [[1511.28,-176.34,-624.91],[0.032971,0.999448,0.003972,-0.00071],[0,-1,-1,0],[0,9E9,9E9,9E9,9E9,9E9]],Work,z10,custom_tool1\WObj:=WObj0;
MoveL [[1521.05,-174.21,-624.92],[0.032971,0.999448,0.003972,-0.00071],[0,-1,-1,0],[0,9E9,9E9,9E9,9E9,9E9]],Work,z10,custom_tool1\WObj:=WObj0;
MoveL [[1530.82,-172.09,-624.94],[0.032971,0.999448,0.003972,-0.00071],[0,-1,-1,0],[0,9E9,9E9,9E9,9E9,9E9]],Work,z10,custom_tool1\WObj:=WObj0;
MoveL [[1540.6,-169.97,-624.96],[0.032971,0.999448,0.003972,-0.00071],[0,-1,-1,0],[0,9E9,9E9,9E9,9E9,9E9]],Work,z10,custom_tool1\WObj:=WObj0;
MoveL [[1550.37,-167.85,-624.97],[0.032971,0.999448,0.003972,-0.00071],[0,-1,-1,0],[0,9E9,9E9,9E9,9E9,9E9]],Work,z10,custom_tool1\WObj:=WObj0;
MoveL [[1560.14,-165.72,-624.99],[0.032971,0.999448,0.003972,-0.00071],[0,-1,-1,0],[0,9E9,9E9,9E9,9E9,9E9]],Work,z10,custom_tool1\WObj:=WObj0;
MoveL [[1569.91,-163.6,-625.01],[0.032971,0.999448,0.003972,-0.00071],[0,-1,-1,0],[0,9E9,9E9,9E9,9E9,9E9]],Work,z10,custom_tool1\WObj:=WObj0;
MoveL [[1579.69,-161.48,-625.02],[0.032971,0.999448,0.003972,-0.00071],[0,-1,-1,0],[0,9E9,9E9,9E9,9E9,9E9]],Work,z10,custom_tool1\WObj:=WObj0;
MoveL [[1589.46,-159.36,-625.04],[0.032971,0.999448,0.003972,-0.00071],[0,-1,-1,0],[0,9E9,9E9,9E9,9E9,9E9]],Work,z10,custom_tool1\WObj:=WObj0;
MoveL [[1599.23,-157.23,-625.05],[0.032971,0.999448,0.003972,-0.00071],[0,-1,-1,0],[0,9E9,9E9,9E9,9E9,9E9]],Work,z10,custom_tool1\WObj:=WObj0;
MoveL [[1609,-155.11,-625.07],[0.032971,0.999448,0.003972,-0.00071],[0,-1,-1,0],[0,9E9,9E9,9E9,9E9,9E9]],Work,z10,custom_tool1\WObj:=WObj0;
MoveL [[1618.77,-152.99,-625.09],[0.032971,0.999448,0.003972,-0.00071],[0,-1,-1,0],[0,9E9,9E9,9E9,9E9,9E9]],Work,z10,custom_tool1\WObj:=WObj0;
MoveL [[1619.17,-157,-625.09],[0.032971,0.999448,0.003972,-0.00071],[0,-1,-1,0],[0,9E9,9E9,9E9,9E9,9E9]],Work,z10,custom_tool1\WObj:=WObj0;
MoveL [[1609.4,-159.12,-625.08],[0.032971,0.999448,0.003972,-0.00071],[0,-1,-1,0],[0,9E9,9E9,9E9,9E9,9E9]],Work,z10,custom_tool1\WObj:=WObj0;
MoveL [[1599.62,-161.24,-625.06],[0.032971,0.999448,0.003972,-0.00071],[0,-1,-1,0],[0,9E9,9E9,9E9,9E9,9E9]],Work,z10,custom_tool1\WObj:=WObj0;
MoveL [[1589.85,-163.36,-625.04],[0.032971,0.999448,0.003972,-0.00071],[0,-1,-1,0],[0,9E9,9E9,9E9,9E9,9E9]],Work,z10,custom_tool1\WObj:=WObj0;
MoveL [[1580.08,-165.49,-625.03],[0.032971,0.999448,0.003972,-0.00071],[0,-1,-1,0],[0,9E9,9E9,9E9,9E9,9E9]],Work,z10,custom_tool1\WObj:=WObj0;
MoveL [[1570.31,-167.61,-625.01],[0.032971,0.999448,0.003972,-0.00071],[0,-1,-1,0],[0,9E9,9E9,9E9,9E9,9E9]],Work,z10,custom_tool1\WObj:=WObj0;
MoveL [[1560.54,-169.73,-624.99],[0.032971,0.999448,0.003972,-0.00071],[0,-1,-1,0],[0,9E9,9E9,9E9,9E9,9E9]],Work,z10,custom_tool1\WObj:=WObj0;
MoveL [[1550.76,-171.85,-624.98],[0.032971,0.999448,0.003972,-0.00071],[0,-1,-1,0],[0,9E9,9E9,9E9,9E9,9E9]],Work,z10,custom_tool1\WObj:=WObj0;
MoveL [[1540.99,-173.98,-624.96],[0.032971,0.999448,0.003972,-0.00071],[0,-1,-1,0],[0,9E9,9E9,9E9,9E9,9E9]],Work,z10,custom_tool1\WObj:=WObj0;
MoveL [[1531.22,-176.1,-624.95],[0.032971,0.999448,0.003972,-0.00071],[0,-1,-1,0],[0,9E9,9E9,9E9,9E9,9E9]],Work,z10,custom_tool1\WObj:=WObj0;
MoveL [[1521.45,-178.22,-624.93],[0.032971,0.999448,0.003972,-0.00071],[0,-1,-1,0],[0,9E9,9E9,9E9,9E9,9E9]],Work,z10,custom_tool1\WObj:=WObj0;
MoveL [[1511.68,-180.34,-624.91],[0.032971,0.999448,0.003972,-0.00071],[0,-1,-1,0],[0,9E9,9E9,9E9,9E9,9E9]],Work,z10,custom_tool1\WObj:=WObj0;
MoveL [[1501.9,-182.47,-624.9],[0.032971,0.999448,0.003972,-0.00071],[0,-1,-1,0],[0,9E9,9E9,9E9,9E9,9E9]],Work,z10,custom_tool1\WObj:=WObj0;
MoveL [[1501.64,-186.62,-624.9],[0.032971,0.999448,0.003972,-0.00071],[0,-1,-1,0],[0,9E9,9E9,9E9,9E9,9E9]],Work,z10,custom_tool1\WObj:=WObj0;
MoveL [[1511.42,-184.49,-624.92],[0.032971,0.999448,0.003972,-0.00071],[0,-1,-1,0],[0,9E9,9E9,9E9,9E9,9E9]],Work,z10,custom_tool1\WObj:=WObj0;
MoveL [[1521.19,-182.37,-624.93],[0.032971,0.999448,0.003972,-0.00071],[0,-1,-1,0],[0,9E9,9E9,9E9,9E9,9E9]],Work,z10,custom_tool1\WObj:=WObj0;
MoveL [[1530.96,-180.25,-624.95],[0.032971,0.999448,0.003972,-0.00071],[0,-1,-1,0],[0,9E9,9E9,9E9,9E9,9E9]],Work,z10,custom_tool1\WObj:=WObj0;
MoveL [[1540.73,-178.13,-624.97],[0.032971,0.999448,0.003972,-0.00071],[0,-1,-1,0],[0,9E9,9E9,9E9,9E9,9E9]],Work,z10,custom_tool1\WObj:=WObj0;
MoveL [[1550.5,-176,-624.98],[0.032971,0.999448,0.003972,-0.00071],[0,-1,-1,0],[0,9E9,9E9,9E9,9E9,9E9]],Work,z10,custom_tool1\WObj:=WObj0;
MoveL [[1560.28,-173.88,-625],[0.032971,0.999448,0.003972,-0.00071],[0,-1,-1,0],[0,9E9,9E9,9E9,9E9,9E9]],Work,z10,custom_tool1\WObj:=WObj0;
MoveL [[1570.05,-171.76,-625.02],[0.032971,0.999448,0.003972,-0.00071],[0,-1,-1,0],[0,9E9,9E9,9E9,9E9,9E9]],Work,z10,custom_tool1\WObj:=WObj0;
MoveL [[1579.82,-169.64,-625.03],[0.032971,0.999448,0.003972,-0.00071],[0,-1,-1,0],[0,9E9,9E9,9E9,9E9,9E9]],Work,z10,custom_tool1\WObj:=WObj0;
MoveL [[1589.59,-167.51,-625.05],[0.032971,0.999448,0.003972,-0.00071],[0,-1,-1,0],[0,9E9,9E9,9E9,9E9,9E9]],Work,z10,custom_tool1\WObj:=WObj0;
MoveL [[1599.36,-165.39,-625.07],[0.032971,0.999448,0.003972,-0.00071],[0,-1,-1,0],[0,9E9,9E9,9E9,9E9,9E9]],Work,z10,custom_tool1\WObj:=WObj0;
MoveL [[1609.14,-163.27,-625.08],[0.032971,0.999448,0.003972,-0.00071],[0,-1,-1,0],[0,9E9,9E9,9E9,9E9,9E9]],Work,z10,custom_tool1\WObj:=WObj0;
MoveL [[1618.91,-161.15,-625.1],[0.032971,0.999448,0.003972,-0.00071],[0,-1,-1,0],[0,9E9,9E9,9E9,9E9,9E9]],Work,z10,custom_tool1\WObj:=WObj0;
MoveL [[1619.3,-165.15,-625.11],[0.032971,0.999448,0.003972,-0.00071],[0,-1,-1,0],[0,9E9,9E9,9E9,9E9,9E9]],Work,z10,custom_tool1\WObj:=WObj0;
MoveL [[1609.53,-167.28,-625.09],[0.032971,0.999448,0.003972,-0.00071],[0,-1,-1,0],[0,9E9,9E9,9E9,9E9,9E9]],Work,z10,custom_tool1\WObj:=WObj0;
MoveL [[1599.76,-169.4,-625.07],[0.032971,0.999448,0.003972,-0.00071],[0,-1,-1,0],[0,9E9,9E9,9E9,9E9,9E9]],Work,z10,custom_tool1\WObj:=WObj0;
MoveL [[1589.99,-171.52,-625.06],[0.032971,0.999448,0.003972,-0.00071],[0,-1,-1,0],[0,9E9,9E9,9E9,9E9,9E9]],Work,z10,custom_tool1\WObj:=WObj0;
MoveL [[1580.22,-173.64,-625.04],[0.032971,0.999448,0.003972,-0.00071],[0,-1,-1,0],[0,9E9,9E9,9E9,9E9,9E9]],Work,z10,custom_tool1\WObj:=WObj0;
MoveL [[1570.44,-175.77,-625.02],[0.032971,0.999448,0.003972,-0.00071],[0,-1,-1,0],[0,9E9,9E9,9E9,9E9,9E9]],Work,z10,custom_tool1\WObj:=WObj0;
MoveL [[1560.67,-177.89,-625.01],[0.032971,0.999448,0.003972,-0.00071],[0,-1,-1,0],[0,9E9,9E9,9E9,9E9,9E9]],Work,z10,custom_tool1\WObj:=WObj0;
MoveL [[1550.9,-180.01,-624.99],[0.032971,0.999448,0.003972,-0.00071],[0,-1,-1,0],[0,9E9,9E9,9E9,9E9,9E9]],Work,z10,custom_tool1\WObj:=WObj0;
MoveL [[1541.13,-182.13,-624.97],[0.032971,0.999448,0.003972,-0.00071],[0,-1,-1,0],[0,9E9,9E9,9E9,9E9,9E9]],Work,z10,custom_tool1\WObj:=WObj0;
MoveL [[1531.36,-184.26,-624.96],[0.032971,0.999448,0.003972,-0.00071],[0,-1,-1,0],[0,9E9,9E9,9E9,9E9,9E9]],Work,z10,custom_tool1\WObj:=WObj0;
MoveL [[1521.58,-186.38,-624.94],[0.032971,0.999448,0.003972,-0.00071],[0,-1,-1,0],[0,9E9,9E9,9E9,9E9,9E9]],Work,z10,custom_tool1\WObj:=WObj0;
MoveL [[1511.81,-188.5,-624.92],[0.032971,0.999448,0.003972,-0.00071],[0,-1,-1,0],[0,9E9,9E9,9E9,9E9,9E9]],Work,z10,custom_tool1\WObj:=WObj0;
MoveL [[1502.04,-190.62,-624.91],[0.032971,0.999448,0.003972,-0.00071],[0,-1,-1,0],[0,9E9,9E9,9E9,9E9,9E9]],Work,z10,custom_tool1\WObj:=WObj0;
MoveL [[1501.78,-194.77,-624.91],[0.032971,0.999448,0.003972,-0.00071],[0,-1,-1,0],[0,9E9,9E9,9E9,9E9,9E9]],Work,z10,custom_tool1\WObj:=WObj0;
MoveL [[1511.55,-192.65,-624.93],[0.032971,0.999448,0.003972,-0.00071],[0,-1,-1,0],[0,9E9,9E9,9E9,9E9,9E9]],Work,z10,custom_tool1\WObj:=WObj0;
MoveL [[1521.32,-190.53,-624.94],[0.032971,0.999448,0.003972,-0.00071],[0,-1,-1,0],[0,9E9,9E9,9E9,9E9,9E9]],Work,z10,custom_tool1\WObj:=WObj0;
MoveL [[1531.09,-188.41,-624.96],[0.032971,0.999448,0.003972,-0.00071],[0,-1,-1,0],[0,9E9,9E9,9E9,9E9,9E9]],Work,z10,custom_tool1\WObj:=WObj0;
MoveL [[1540.87,-186.28,-624.98],[0.032971,0.999448,0.003972,-0.00071],[0,-1,-1,0],[0,9E9,9E9,9E9,9E9,9E9]],Work,z10,custom_tool1\WObj:=WObj0;
MoveL [[1550.64,-184.16,-624.99],[0.032971,0.999448,0.003972,-0.00071],[0,-1,-1,0],[0,9E9,9E9,9E9,9E9,9E9]],Work,z10,custom_tool1\WObj:=WObj0;
MoveL [[1560.41,-182.04,-625.01],[0.032971,0.999448,0.003972,-0.00071],[0,-1,-1,0],[0,9E9,9E9,9E9,9E9,9E9]],Work,z10,custom_tool1\WObj:=WObj0;
MoveL [[1570.18,-179.92,-625.03],[0.032971,0.999448,0.003972,-0.00071],[0,-1,-1,0],[0,9E9,9E9,9E9,9E9,9E9]],Work,z10,custom_tool1\WObj:=WObj0;
MoveL [[1579.95,-177.79,-625.04],[0.032971,0.999448,0.003972,-0.00071],[0,-1,-1,0],[0,9E9,9E9,9E9,9E9,9E9]],Work,z10,custom_tool1\WObj:=WObj0;
MoveL [[1589.73,-175.67,-625.06],[0.032971,0.999448,0.003972,-0.00071],[0,-1,-1,0],[0,9E9,9E9,9E9,9E9,9E9]],Work,z10,custom_tool1\WObj:=WObj0;
MoveL [[1599.5,-173.55,-625.08],[0.032971,0.999448,0.003972,-0.00071],[0,-1,-1,0],[0,9E9,9E9,9E9,9E9,9E9]],Work,z10,custom_tool1\WObj:=WObj0;
MoveL [[1609.27,-171.43,-625.09],[0.032971,0.999448,0.003972,-0.00071],[0,-1,-1,0],[0,9E9,9E9,9E9,9E9,9E9]],Work,z10,custom_tool1\WObj:=WObj0;
MoveL [[1619.04,-169.3,-625.11],[0.032971,0.999448,0.003972,-0.00071],[0,-1,-1,0],[0,9E9,9E9,9E9,9E9,9E9]],Work,z10,custom_tool1\WObj:=WObj0;
MoveL [[1619.44,-173.31,-625.12],[0.032971,0.999448,0.003972,-0.00071],[0,-1,-1,0],[0,9E9,9E9,9E9,9E9,9E9]],Work,z10,custom_tool1\WObj:=WObj0;
MoveL [[1609.67,-175.43,-625.1],[0.032971,0.999448,0.003972,-0.00071],[0,-1,-1,0],[0,9E9,9E9,9E9,9E9,9E9]],Work,z10,custom_tool1\WObj:=WObj0;
MoveL [[1599.9,-177.56,-625.08],[0.032971,0.999448,0.003972,-0.00071],[0,-1,-1,0],[0,9E9,9E9,9E9,9E9,9E9]],Work,z10,custom_tool1\WObj:=WObj0;
MoveL [[1590.12,-179.68,-625.07],[0.032971,0.999448,0.003972,-0.00071],[0,-1,-1,0],[0,9E9,9E9,9E9,9E9,9E9]],Work,z10,custom_tool1\WObj:=WObj0;
MoveL [[1580.35,-181.8,-625.05],[0.032971,0.999448,0.003972,-0.00071],[0,-1,-1,0],[0,9E9,9E9,9E9,9E9,9E9]],Work,z10,custom_tool1\WObj:=WObj0;
MoveL [[1570.58,-183.92,-625.03],[0.032971,0.999448,0.003972,-0.00071],[0,-1,-1,0],[0,9E9,9E9,9E9,9E9,9E9]],Work,z10,custom_tool1\WObj:=WObj0;
MoveL [[1560.81,-186.05,-625.02],[0.032971,0.999448,0.003972,-0.00071],[0,-1,-1,0],[0,9E9,9E9,9E9,9E9,9E9]],Work,z10,custom_tool1\WObj:=WObj0;
MoveL [[1551.03,-188.17,-625],[0.032971,0.999448,0.003972,-0.00071],[0,-1,-1,0],[0,9E9,9E9,9E9,9E9,9E9]],Work,z10,custom_tool1\WObj:=WObj0;
MoveL [[1541.26,-190.29,-624.98],[0.032971,0.999448,0.003972,-0.00071],[0,-1,-1,0],[0,9E9,9E9,9E9,9E9,9E9]],Work,z10,custom_tool1\WObj:=WObj0;
MoveL [[1531.49,-192.41,-624.97],[0.032971,0.999448,0.003972,-0.00071],[0,-1,-1,0],[0,9E9,9E9,9E9,9E9,9E9]],Work,z10,custom_tool1\WObj:=WObj0;
MoveL [[1521.72,-194.54,-624.95],[0.032971,0.999448,0.003972,-0.00071],[0,-1,-1,0],[0,9E9,9E9,9E9,9E9,9E9]],Work,z10,custom_tool1\WObj:=WObj0;
MoveL [[1511.95,-196.66,-624.93],[0.032971,0.999448,0.003972,-0.00071],[0,-1,-1,0],[0,9E9,9E9,9E9,9E9,9E9]],Work,z10,custom_tool1\WObj:=WObj0;
MoveL [[1502.17,-198.78,-624.92],[0.032971,0.999448,0.003972,-0.00071],[0,-1,-1,0],[0,9E9,9E9,9E9,9E9,9E9]],Work,z10,custom_tool1\WObj:=WObj0;
MoveL [[1501.91,-202.93,-624.92],[0.032971,0.999448,0.003972,-0.00071],[0,-1,-1,0],[0,9E9,9E9,9E9,9E9,9E9]],Work,z10,custom_tool1\WObj:=WObj0;
MoveL [[1511.68,-200.81,-624.94],[0.032971,0.999448,0.003972,-0.00071],[0,-1,-1,0],[0,9E9,9E9,9E9,9E9,9E9]],Work,z10,custom_tool1\WObj:=WObj0;
MoveL [[1521.46,-198.69,-624.96],[0.032971,0.999448,0.003972,-0.00071],[0,-1,-1,0],[0,9E9,9E9,9E9,9E9,9E9]],Work,z10,custom_tool1\WObj:=WObj0;
MoveL [[1531.23,-196.56,-624.97],[0.032971,0.999448,0.003972,-0.00071],[0,-1,-1,0],[0,9E9,9E9,9E9,9E9,9E9]],Work,z10,custom_tool1\WObj:=WObj0;
MoveL [[1541,-194.44,-624.99],[0.032971,0.999448,0.003972,-0.00071],[0,-1,-1,0],[0,9E9,9E9,9E9,9E9,9E9]],Work,z10,custom_tool1\WObj:=WObj0;
MoveL [[1550.77,-192.32,-625.01],[0.032971,0.999448,0.003972,-0.00071],[0,-1,-1,0],[0,9E9,9E9,9E9,9E9,9E9]],Work,z10,custom_tool1\WObj:=WObj0;
MoveL [[1560.54,-190.2,-625.02],[0.032971,0.999448,0.003972,-0.00071],[0,-1,-1,0],[0,9E9,9E9,9E9,9E9,9E9]],Work,z10,custom_tool1\WObj:=WObj0;
MoveL [[1570.32,-188.07,-625.04],[0.032971,0.999448,0.003972,-0.00071],[0,-1,-1,0],[0,9E9,9E9,9E9,9E9,9E9]],Work,z10,custom_tool1\WObj:=WObj0;
MoveL [[1580.09,-185.95,-625.06],[0.032971,0.999448,0.003972,-0.00071],[0,-1,-1,0],[0,9E9,9E9,9E9,9E9,9E9]],Work,z10,custom_tool1\WObj:=WObj0;
MoveL [[1589.86,-183.83,-625.07],[0.032971,0.999448,0.003972,-0.00071],[0,-1,-1,0],[0,9E9,9E9,9E9,9E9,9E9]],Work,z10,custom_tool1\WObj:=WObj0;
MoveL [[1599.63,-181.71,-625.09],[0.032971,0.999448,0.003972,-0.00071],[0,-1,-1,0],[0,9E9,9E9,9E9,9E9,9E9]],Work,z10,custom_tool1\WObj:=WObj0;
MoveL [[1609.41,-179.58,-625.11],[0.032971,0.999448,0.003972,-0.00071],[0,-1,-1,0],[0,9E9,9E9,9E9,9E9,9E9]],Work,z10,custom_tool1\WObj:=WObj0;
MoveL [[1619.18,-177.46,-625.12],[0.032971,0.999448,0.003972,-0.00071],[0,-1,-1,0],[0,9E9,9E9,9E9,9E9,9E9]],Work,z10,custom_tool1\WObj:=WObj0;
MoveL [[1619.57,-181.47,-625.13],[0.032971,0.999448,0.003972,-0.00071],[0,-1,-1,0],[0,9E9,9E9,9E9,9E9,9E9]],Work,z10,custom_tool1\WObj:=WObj0;
MoveL [[1609.8,-183.59,-625.11],[0.032971,0.999448,0.003972,-0.00071],[0,-1,-1,0],[0,9E9,9E9,9E9,9E9,9E9]],Work,z10,custom_tool1\WObj:=WObj0;
MoveL [[1600.03,-185.71,-625.1],[0.032971,0.999448,0.003972,-0.00071],[0,-1,-1,0],[0,9E9,9E9,9E9,9E9,9E9]],Work,z10,custom_tool1\WObj:=WObj0;
MoveL [[1590.26,-187.84,-625.08],[0.032971,0.999448,0.003972,-0.00071],[0,-1,-1,0],[0,9E9,9E9,9E9,9E9,9E9]],Work,z10,custom_tool1\WObj:=WObj0;
MoveL [[1580.49,-189.96,-625.06],[0.032971,0.999448,0.003972,-0.00071],[0,-1,-1,0],[0,9E9,9E9,9E9,9E9,9E9]],Work,z10,custom_tool1\WObj:=WObj0;
MoveL [[1570.71,-192.08,-625.05],[0.032971,0.999448,0.003972,-0.00071],[0,-1,-1,0],[0,9E9,9E9,9E9,9E9,9E9]],Work,z10,custom_tool1\WObj:=WObj0;
MoveL [[1560.94,-194.2,-625.03],[0.032971,0.999448,0.003972,-0.00071],[0,-1,-1,0],[0,9E9,9E9,9E9,9E9,9E9]],Work,z10,custom_tool1\WObj:=WObj0;
MoveL [[1551.17,-196.33,-625.01],[0.032971,0.999448,0.003972,-0.00071],[0,-1,-1,0],[0,9E9,9E9,9E9,9E9,9E9]],Work,z10,custom_tool1\WObj:=WObj0;
MoveL [[1541.4,-198.45,-625],[0.032971,0.999448,0.003972,-0.00071],[0,-1,-1,0],[0,9E9,9E9,9E9,9E9,9E9]],Work,z10,custom_tool1\WObj:=WObj0;
MoveL [[1531.62,-200.57,-624.98],[0.032971,0.999448,0.003972,-0.00071],[0,-1,-1,0],[0,9E9,9E9,9E9,9E9,9E9]],Work,z10,custom_tool1\WObj:=WObj0;
MoveL [[1521.85,-202.69,-624.96],[0.032971,0.999448,0.003972,-0.00071],[0,-1,-1,0],[0,9E9,9E9,9E9,9E9,9E9]],Work,z10,custom_tool1\WObj:=WObj0;
MoveL [[1512.08,-204.82,-624.95],[0.032971,0.999448,0.003972,-0.00071],[0,-1,-1,0],[0,9E9,9E9,9E9,9E9,9E9]],Work,z10,custom_tool1\WObj:=WObj0;
MoveL [[1502.31,-206.94,-624.93],[0.032971,0.999448,0.003972,-0.00071],[0,-1,-1,0],[0,9E9,9E9,9E9,9E9,9E9]],Work,z10,custom_tool1\WObj:=WObj0;
MoveL [[1502.05,-211.09,-624.93],[0.032971,0.999448,0.003972,-0.00071],[0,-1,-1,0],[0,9E9,9E9,9E9,9E9,9E9]],Work,z10,custom_tool1\WObj:=WObj0;
MoveL [[1511.82,-208.97,-624.95],[0.032971,0.999448,0.003972,-0.00071],[0,-1,-1,0],[0,9E9,9E9,9E9,9E9,9E9]],Work,z10,custom_tool1\WObj:=WObj0;
MoveL [[1521.59,-206.84,-624.97],[0.032971,0.999448,0.003972,-0.00071],[0,-1,-1,0],[0,9E9,9E9,9E9,9E9,9E9]],Work,z10,custom_tool1\WObj:=WObj0;
MoveL [[1531.36,-204.72,-624.98],[0.032971,0.999448,0.003972,-0.00071],[0,-1,-1,0],[0,9E9,9E9,9E9,9E9,9E9]],Work,z10,custom_tool1\WObj:=WObj0;
MoveL [[1541.13,-202.6,-625],[0.032971,0.999448,0.003972,-0.00071],[0,-1,-1,0],[0,9E9,9E9,9E9,9E9,9E9]],Work,z10,custom_tool1\WObj:=WObj0;
MoveL [[1550.91,-200.48,-625.02],[0.032971,0.999448,0.003972,-0.00071],[0,-1,-1,0],[0,9E9,9E9,9E9,9E9,9E9]],Work,z10,custom_tool1\WObj:=WObj0;
MoveL [[1560.68,-198.35,-625.03],[0.032971,0.999448,0.003972,-0.00071],[0,-1,-1,0],[0,9E9,9E9,9E9,9E9,9E9]],Work,z10,custom_tool1\WObj:=WObj0;
MoveL [[1570.45,-196.23,-625.05],[0.032971,0.999448,0.003972,-0.00071],[0,-1,-1,0],[0,9E9,9E9,9E9,9E9,9E9]],Work,z10,custom_tool1\WObj:=WObj0;
MoveL [[1580.22,-194.11,-625.07],[0.032971,0.999448,0.003972,-0.00071],[0,-1,-1,0],[0,9E9,9E9,9E9,9E9,9E9]],Work,z10,custom_tool1\WObj:=WObj0;
MoveL [[1590,-191.99,-625.08],[0.032971,0.999448,0.003972,-0.00071],[0,-1,-1,0],[0,9E9,9E9,9E9,9E9,9E9]],Work,z10,custom_tool1\WObj:=WObj0;
MoveL [[1599.77,-189.86,-625.1],[0.032971,0.999448,0.003972,-0.00071],[0,-1,-1,0],[0,9E9,9E9,9E9,9E9,9E9]],Work,z10,custom_tool1\WObj:=WObj0;
MoveL [[1609.54,-187.74,-625.12],[0.032971,0.999448,0.003972,-0.00071],[0,-1,-1,0],[0,9E9,9E9,9E9,9E9,9E9]],Work,z10,custom_tool1\WObj:=WObj0;
MoveL [[1619.31,-185.62,-625.13],[0.032971,0.999448,0.003972,-0.00071],[0,-1,-1,0],[0,9E9,9E9,9E9,9E9,9E9]],Work,z10,custom_tool1\WObj:=WObj0;
MoveL [[1619.71,-189.63,-625.14],[0.032971,0.999448,0.003972,-0.00071],[0,-1,-1,0],[0,9E9,9E9,9E9,9E9,9E9]],Work,z10,custom_tool1\WObj:=WObj0;
MoveL [[1609.94,-191.75,-625.12],[0.032971,0.999448,0.003972,-0.00071],[0,-1,-1,0],[0,9E9,9E9,9E9,9E9,9E9]],Work,z10,custom_tool1\WObj:=WObj0;
MoveL [[1600.16,-193.87,-625.11],[0.032971,0.999448,0.003972,-0.00071],[0,-1,-1,0],[0,9E9,9E9,9E9,9E9,9E9]],Work,z10,custom_tool1\WObj:=WObj0;
MoveL [[1590.39,-195.99,-625.09],[0.032971,0.999448,0.003972,-0.00071],[0,-1,-1,0],[0,9E9,9E9,9E9,9E9,9E9]],Work,z10,custom_tool1\WObj:=WObj0;
MoveL [[1580.62,-198.12,-625.07],[0.032971,0.999448,0.003972,-0.00071],[0,-1,-1,0],[0,9E9,9E9,9E9,9E9,9E9]],Work,z10,custom_tool1\WObj:=WObj0;
MoveL [[1570.85,-200.24,-625.06],[0.032971,0.999448,0.003972,-0.00071],[0,-1,-1,0],[0,9E9,9E9,9E9,9E9,9E9]],Work,z10,custom_tool1\WObj:=WObj0;
MoveL [[1561.08,-202.36,-625.04],[0.032971,0.999448,0.003972,-0.00071],[0,-1,-1,0],[0,9E9,9E9,9E9,9E9,9E9]],Work,z10,custom_tool1\WObj:=WObj0;
MoveL [[1551.3,-204.48,-625.02],[0.032971,0.999448,0.003972,-0.00071],[0,-1,-1,0],[0,9E9,9E9,9E9,9E9,9E9]],Work,z10,custom_tool1\WObj:=WObj0;
MoveL [[1541.53,-206.61,-625.01],[0.032971,0.999448,0.003972,-0.00071],[0,-1,-1,0],[0,9E9,9E9,9E9,9E9,9E9]],Work,z10,custom_tool1\WObj:=WObj0;
MoveL [[1531.76,-208.73,-624.99],[0.032971,0.999448,0.003972,-0.00071],[0,-1,-1,0],[0,9E9,9E9,9E9,9E9,9E9]],Work,z10,custom_tool1\WObj:=WObj0;
MoveL [[1521.99,-210.85,-624.97],[0.032971,0.999448,0.003972,-0.00071],[0,-1,-1,0],[0,9E9,9E9,9E9,9E9,9E9]],Work,z10,custom_tool1\WObj:=WObj0;
MoveL [[1512.21,-212.97,-624.96],[0.032971,0.999448,0.003972,-0.00071],[0,-1,-1,0],[0,9E9,9E9,9E9,9E9,9E9]],Work,z10,custom_tool1\WObj:=WObj0;
MoveL [[1502.44,-215.1,-624.94],[0.032971,0.999448,0.003972,-0.00071],[0,-1,-1,0],[0,9E9,9E9,9E9,9E9,9E9]],Work,z10,custom_tool1\WObj:=WObj0;
MoveL [[1502.18,-219.25,-624.95],[0.032971,0.999448,0.003972,-0.00071],[0,-1,-1,0],[0,9E9,9E9,9E9,9E9,9E9]],Work,z10,custom_tool1\WObj:=WObj0;
MoveL [[1511.95,-217.12,-624.96],[0.032971,0.999448,0.003972,-0.00071],[0,-1,-1,0],[0,9E9,9E9,9E9,9E9,9E9]],Work,z10,custom_tool1\WObj:=WObj0;
MoveL [[1521.73,-215,-624.98],[0.032971,0.999448,0.003972,-0.00071],[0,-1,-1,0],[0,9E9,9E9,9E9,9E9,9E9]],Work,z10,custom_tool1\WObj:=WObj0;
MoveL [[1531.5,-212.88,-625],[0.032971,0.999448,0.003972,-0.00071],[0,-1,-1,0],[0,9E9,9E9,9E9,9E9,9E9]],Work,z10,custom_tool1\WObj:=WObj0;
MoveL [[1541.27,-210.76,-625.01],[0.032971,0.999448,0.003972,-0.00071],[0,-1,-1,0],[0,9E9,9E9,9E9,9E9,9E9]],Work,z10,custom_tool1\WObj:=WObj0;
MoveL [[1551.04,-208.63,-625.03],[0.032971,0.999448,0.003972,-0.00071],[0,-1,-1,0],[0,9E9,9E9,9E9,9E9,9E9]],Work,z10,custom_tool1\WObj:=WObj0;
MoveL [[1560.81,-206.51,-625.05],[0.032971,0.999448,0.003972,-0.00071],[0,-1,-1,0],[0,9E9,9E9,9E9,9E9,9E9]],Work,z10,custom_tool1\WObj:=WObj0;
MoveL [[1570.59,-204.39,-625.06],[0.032971,0.999448,0.003972,-0.00071],[0,-1,-1,0],[0,9E9,9E9,9E9,9E9,9E9]],Work,z10,custom_tool1\WObj:=WObj0;
MoveL [[1580.36,-202.27,-625.08],[0.032971,0.999448,0.003972,-0.00071],[0,-1,-1,0],[0,9E9,9E9,9E9,9E9,9E9]],Work,z10,custom_tool1\WObj:=WObj0;
MoveL [[1590.13,-200.14,-625.1],[0.032971,0.999448,0.003972,-0.00071],[0,-1,-1,0],[0,9E9,9E9,9E9,9E9,9E9]],Work,z10,custom_tool1\WObj:=WObj0;
MoveL [[1599.9,-198.02,-625.11],[0.032971,0.999448,0.003972,-0.00071],[0,-1,-1,0],[0,9E9,9E9,9E9,9E9,9E9]],Work,z10,custom_tool1\WObj:=WObj0;
MoveL [[1609.67,-195.9,-625.13],[0.032971,0.999448,0.003972,-0.00071],[0,-1,-1,0],[0,9E9,9E9,9E9,9E9,9E9]],Work,z10,custom_tool1\WObj:=WObj0;
MoveL [[1619.45,-193.78,-625.14],[0.032971,0.999448,0.003972,-0.00071],[0,-1,-1,0],[0,9E9,9E9,9E9,9E9,9E9]],Work,z10,custom_tool1\WObj:=WObj0;
MoveL [[1619.84,-197.78,-625.15],[0.032971,0.999448,0.003972,-0.00071],[0,-1,-1,0],[0,9E9,9E9,9E9,9E9,9E9]],Work,z10,custom_tool1\WObj:=WObj0;
MoveL [[1610.07,-199.91,-625.13],[0.032971,0.999448,0.003972,-0.00071],[0,-1,-1,0],[0,9E9,9E9,9E9,9E9,9E9]],Work,z10,custom_tool1\WObj:=WObj0;
MoveL [[1600.3,-202.03,-625.12],[0.032971,0.999448,0.003972,-0.00071],[0,-1,-1,0],[0,9E9,9E9,9E9,9E9,9E9]],Work,z10,custom_tool1\WObj:=WObj0;
MoveL [[1590.53,-204.15,-625.1],[0.032971,0.999448,0.003972,-0.00071],[0,-1,-1,0],[0,9E9,9E9,9E9,9E9,9E9]],Work,z10,custom_tool1\WObj:=WObj0;
MoveL [[1580.75,-206.27,-625.08],[0.032971,0.999448,0.003972,-0.00071],[0,-1,-1,0],[0,9E9,9E9,9E9,9E9,9E9]],Work,z10,custom_tool1\WObj:=WObj0;
MoveL [[1570.98,-208.4,-625.07],[0.032971,0.999448,0.003972,-0.00071],[0,-1,-1,0],[0,9E9,9E9,9E9,9E9,9E9]],Work,z10,custom_tool1\WObj:=WObj0;
MoveL [[1561.21,-210.52,-625.05],[0.032971,0.999448,0.003972,-0.00071],[0,-1,-1,0],[0,9E9,9E9,9E9,9E9,9E9]],Work,z10,custom_tool1\WObj:=WObj0;
MoveL [[1551.44,-212.64,-625.03],[0.032971,0.999448,0.003972,-0.00071],[0,-1,-1,0],[0,9E9,9E9,9E9,9E9,9E9]],Work,z10,custom_tool1\WObj:=WObj0;
MoveL [[1541.67,-214.76,-625.02],[0.032971,0.999448,0.003972,-0.00071],[0,-1,-1,0],[0,9E9,9E9,9E9,9E9,9E9]],Work,z10,custom_tool1\WObj:=WObj0;
MoveL [[1531.89,-216.89,-625],[0.032971,0.999448,0.003972,-0.00071],[0,-1,-1,0],[0,9E9,9E9,9E9,9E9,9E9]],Work,z10,custom_tool1\WObj:=WObj0;
MoveL [[1522.12,-219.01,-624.99],[0.032971,0.999448,0.003972,-0.00071],[0,-1,-1,0],[0,9E9,9E9,9E9,9E9,9E9]],Work,z10,custom_tool1\WObj:=WObj0;
MoveL [[1512.35,-221.13,-624.97],[0.032971,0.999448,0.003972,-0.00071],[0,-1,-1,0],[0,9E9,9E9,9E9,9E9,9E9]],Work,z10,custom_tool1\WObj:=WObj0;
MoveL [[1502.58,-223.25,-624.95],[0.032971,0.999448,0.003972,-0.00071],[0,-1,-1,0],[0,9E9,9E9,9E9,9E9,9E9]],Work,z10,custom_tool1\WObj:=WObj0;
MoveL [[1502.32,-227.4,-624.96],[0.032971,0.999448,0.003972,-0.00071],[0,-1,-1,0],[0,9E9,9E9,9E9,9E9,9E9]],Work,z10,custom_tool1\WObj:=WObj0;
MoveL [[1512.09,-225.28,-624.97],[0.032971,0.999448,0.003972,-0.00071],[0,-1,-1,0],[0,9E9,9E9,9E9,9E9,9E9]],Work,z10,custom_tool1\WObj:=WObj0;
MoveL [[1521.86,-223.16,-624.99],[0.032971,0.999448,0.003972,-0.00071],[0,-1,-1,0],[0,9E9,9E9,9E9,9E9,9E9]],Work,z10,custom_tool1\WObj:=WObj0;
MoveL [[1531.63,-221.04,-625.01],[0.032971,0.999448,0.003972,-0.00071],[0,-1,-1,0],[0,9E9,9E9,9E9,9E9,9E9]],Work,z10,custom_tool1\WObj:=WObj0;
MoveL [[1541.4,-218.91,-625.02],[0.032971,0.999448,0.003972,-0.00071],[0,-1,-1,0],[0,9E9,9E9,9E9,9E9,9E9]],Work,z10,custom_tool1\WObj:=WObj0;
MoveL [[1551.18,-216.79,-625.04],[0.032971,0.999448,0.003972,-0.00071],[0,-1,-1,0],[0,9E9,9E9,9E9,9E9,9E9]],Work,z10,custom_tool1\WObj:=WObj0;
MoveL [[1560.95,-214.67,-625.06],[0.032971,0.999448,0.003972,-0.00071],[0,-1,-1,0],[0,9E9,9E9,9E9,9E9,9E9]],Work,z10,custom_tool1\WObj:=WObj0;
MoveL [[1570.72,-212.55,-625.07],[0.032971,0.999448,0.003972,-0.00071],[0,-1,-1,0],[0,9E9,9E9,9E9,9E9,9E9]],Work,z10,custom_tool1\WObj:=WObj0;
MoveL [[1580.49,-210.42,-625.09],[0.032971,0.999448,0.003972,-0.00071],[0,-1,-1,0],[0,9E9,9E9,9E9,9E9,9E9]],Work,z10,custom_tool1\WObj:=WObj0;
MoveL [[1590.26,-208.3,-625.11],[0.032971,0.999448,0.003972,-0.00071],[0,-1,-1,0],[0,9E9,9E9,9E9,9E9,9E9]],Work,z10,custom_tool1\WObj:=WObj0;
MoveL [[1600.04,-206.18,-625.12],[0.032971,0.999448,0.003972,-0.00071],[0,-1,-1,0],[0,9E9,9E9,9E9,9E9,9E9]],Work,z10,custom_tool1\WObj:=WObj0;
MoveL [[1609.81,-204.06,-625.14],[0.032971,0.999448,0.003972,-0.00071],[0,-1,-1,0],[0,9E9,9E9,9E9,9E9,9E9]],Work,z10,custom_tool1\WObj:=WObj0;
MoveL [[1619.58,-201.93,-625.16],[0.032971,0.999448,0.003972,-0.00071],[0,-1,-1,0],[0,9E9,9E9,9E9,9E9,9E9]],Work,z10,custom_tool1\WObj:=WObj0;
MoveL [[1619.98,-205.94,-625.16],[0.032971,0.999448,0.003972,-0.00071],[0,-1,-1,0],[0,9E9,9E9,9E9,9E9,9E9]],Work,z10,custom_tool1\WObj:=WObj0;
MoveL [[1610.21,-208.06,-625.15],[0.032971,0.999448,0.003972,-0.00071],[0,-1,-1,0],[0,9E9,9E9,9E9,9E9,9E9]],Work,z10,custom_tool1\WObj:=WObj0;
MoveL [[1600.43,-210.19,-625.13],[0.032971,0.999448,0.003972,-0.00071],[0,-1,-1,0],[0,9E9,9E9,9E9,9E9,9E9]],Work,z10,custom_tool1\WObj:=WObj0;
MoveL [[1590.66,-212.31,-625.11],[0.032971,0.999448,0.003972,-0.00071],[0,-1,-1,0],[0,9E9,9E9,9E9,9E9,9E9]],Work,z10,custom_tool1\WObj:=WObj0;
MoveL [[1580.89,-214.43,-625.1],[0.032971,0.999448,0.003972,-0.00071],[0,-1,-1,0],[0,9E9,9E9,9E9,9E9,9E9]],Work,z10,custom_tool1\WObj:=WObj0;
MoveL [[1571.12,-216.55,-625.08],[0.032971,0.999448,0.003972,-0.00071],[0,-1,-1,0],[0,9E9,9E9,9E9,9E9,9E9]],Work,z10,custom_tool1\WObj:=WObj0;
MoveL [[1561.34,-218.68,-625.06],[0.032971,0.999448,0.003972,-0.00071],[0,-1,-1,0],[0,9E9,9E9,9E9,9E9,9E9]],Work,z10,custom_tool1\WObj:=WObj0;
MoveL [[1551.57,-220.8,-625.05],[0.032971,0.999448,0.003972,-0.00071],[0,-1,-1,0],[0,9E9,9E9,9E9,9E9,9E9]],Work,z10,custom_tool1\WObj:=WObj0;
MoveL [[1541.8,-222.92,-625.03],[0.032971,0.999448,0.003972,-0.00071],[0,-1,-1,0],[0,9E9,9E9,9E9,9E9,9E9]],Work,z10,custom_tool1\WObj:=WObj0;
MoveL [[1532.03,-225.04,-625.01],[0.032971,0.999448,0.003972,-0.00071],[0,-1,-1,0],[0,9E9,9E9,9E9,9E9,9E9]],Work,z10,custom_tool1\WObj:=WObj0;
MoveL [[1522.26,-227.17,-625],[0.032971,0.999448,0.003972,-0.00071],[0,-1,-1,0],[0,9E9,9E9,9E9,9E9,9E9]],Work,z10,custom_tool1\WObj:=WObj0;
MoveL [[1512.48,-229.29,-624.98],[0.032971,0.999448,0.003972,-0.00071],[0,-1,-1,0],[0,9E9,9E9,9E9,9E9,9E9]],Work,z10,custom_tool1\WObj:=WObj0;
MoveL [[1502.71,-231.41,-624.96],[0.032971,0.999448,0.003972,-0.00071],[0,-1,-1,0],[0,9E9,9E9,9E9,9E9,9E9]],Work,z10,custom_tool1\WObj:=WObj0;
MoveL [[1502.45,-235.56,-624.97],[0.032971,0.999448,0.003972,-0.00071],[0,-1,-1,0],[0,9E9,9E9,9E9,9E9,9E9]],Work,z10,custom_tool1\WObj:=WObj0;
MoveL [[1512.22,-233.44,-624.99],[0.032971,0.999448,0.003972,-0.00071],[0,-1,-1,0],[0,9E9,9E9,9E9,9E9,9E9]],Work,z10,custom_tool1\WObj:=WObj0;
MoveL [[1521.99,-231.32,-625],[0.032971,0.999448,0.003972,-0.00071],[0,-1,-1,0],[0,9E9,9E9,9E9,9E9,9E9]],Work,z10,custom_tool1\WObj:=WObj0;
MoveL [[1531.77,-229.19,-625.02],[0.032971,0.999448,0.003972,-0.00071],[0,-1,-1,0],[0,9E9,9E9,9E9,9E9,9E9]],Work,z10,custom_tool1\WObj:=WObj0;
MoveL [[1541.54,-227.07,-625.03],[0.032971,0.999448,0.003972,-0.00071],[0,-1,-1,0],[0,9E9,9E9,9E9,9E9,9E9]],Work,z10,custom_tool1\WObj:=WObj0;
MoveL [[1551.31,-224.95,-625.05],[0.032971,0.999448,0.003972,-0.00071],[0,-1,-1,0],[0,9E9,9E9,9E9,9E9,9E9]],Work,z10,custom_tool1\WObj:=WObj0;
MoveL [[1561.08,-222.83,-625.07],[0.032971,0.999448,0.003972,-0.00071],[0,-1,-1,0],[0,9E9,9E9,9E9,9E9,9E9]],Work,z10,custom_tool1\WObj:=WObj0;
MoveL [[1570.85,-220.7,-625.08],[0.032971,0.999448,0.003972,-0.00071],[0,-1,-1,0],[0,9E9,9E9,9E9,9E9,9E9]],Work,z10,custom_tool1\WObj:=WObj0;
